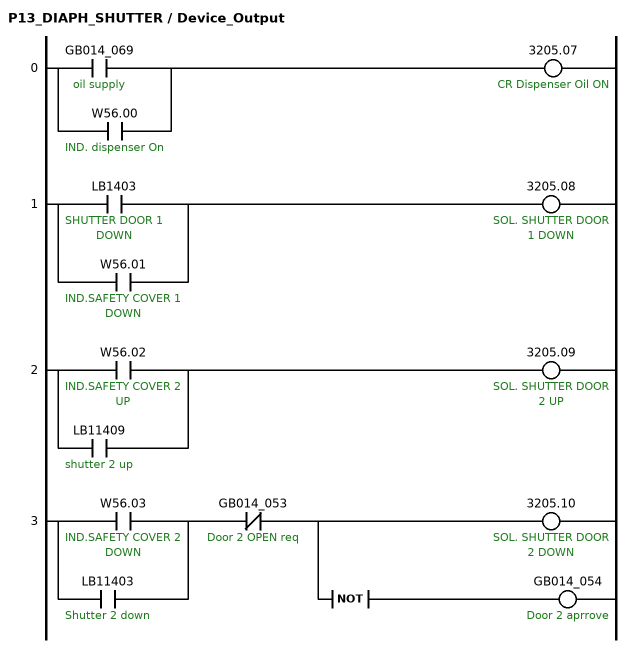
; [picture p168: P13_DIAPH_SHUTTER / Device_Output, rungs 0-3]
; rung 0
LD GB014_069  ; oil supply
OR W56.00  ; IND. dispenser On
OUT 3205.07  ; CR Dispenser Oil ON
; rung 1
LD LB1403  ; SHUTTER DOOR 1 DOWN
OR W56.01  ; IND.SAFETY COVER 1 DOWN
OUT 3205.08  ; SOL. SHUTTER DOOR 1 DOWN
; rung 2
LD W56.02  ; IND.SAFETY COVER 2 UP
OR LB11409  ; shutter 2 up
OUT 3205.09  ; SOL. SHUTTER DOOR 2 UP
; rung 3
LD W56.03  ; IND.SAFETY COVER 2 DOWN
OR LB11403  ; Shutter 2 down
ANDNOT GB014_053  ; Door 2 OPEN req
OUT 3205.10  ; SOL. SHUTTER DOOR 2 DOWN
NOT(520)
OUT GB014_054  ; Door 2 aprrove

### Section station_Output

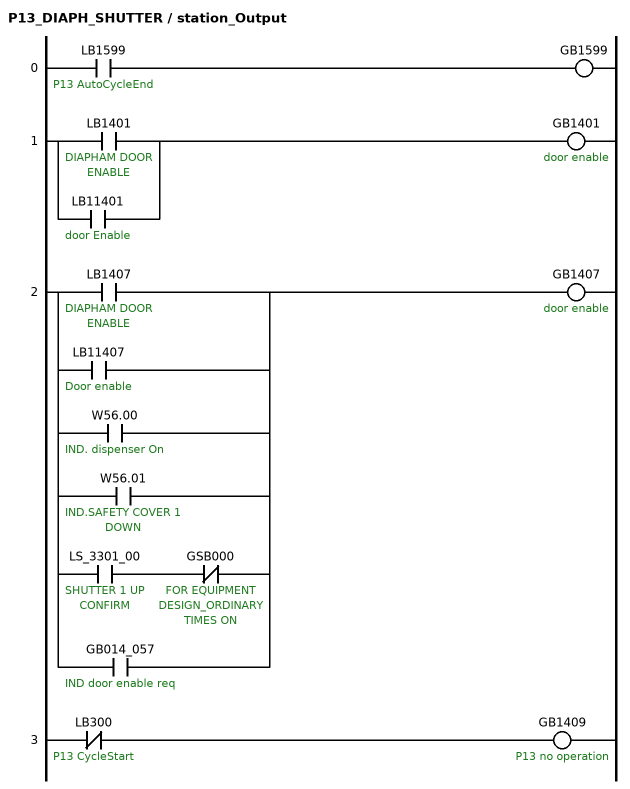
; rung 0
LD LB1599  ; P13 AutoCycleEnd
OUT GB1599
; rung 1
LD LB1401  ; DIAPHAM DOOR ENABLE
OR LB11401  ; door Enable
OUT GB1401  ; door enable
; rung 2
LD LB1407  ; DIAPHAM DOOR ENABLE
OR LB11407  ; Door enable
OR W56.00  ; IND. dispenser On
OR W56.01  ; IND.SAFETY COVER 1 DOWN
LD LS_3301_00  ; SHUTTER 1 UP CONFIRM
ANDNOT GSB000  ; FOR EQUIPMENT DESIGN_ORDINARY TIMES ON
ORLD
OR GB014_057  ; IND door enable req
OUT GB1407  ; door enable
; rung 3
LDNOT LB300  ; P13 CycleStart
OUT GB1409  ; P13 no operation

### Section END
; rung 0
END(001)

## Program P14_DIAPH_LOADER (cyclic task 4)
Local symbols
Disch_last_work E0_16.01 BOOL
Disch_last_work_operation_memory E0_16.02 BOOL
GB014_055 E0_45.06 BOOL  ; DOOR 2 OPEN req
GB014_056 E0_44.11 BOOL  ; IND door enable req
GB014_067 E0_42.12 BOOL  ; vacuum 1start
LB1000 E0_16.03 BOOL  ; AUTO START BEGIN
LB14234 E0_49.14 BOOL  ; oil supply motion
LB14235 E0_49.15 BOOL  ; oil supply finish
LB1600 E0_16.04 BOOL  ; AUTO START BEGIN
LB1601 E0_16.05 BOOL  ; 1EC3 FORWARD START
LB1601_1 E0_44.00 BOOL  ; EC4 backward
LB1601_12 E0_45.03 BOOL  ; Door 2 open req
LB1602 E0_16.06 BOOL  ; 1EC3 FORWARD START COMP
LB1602_1 E0_44.01 BOOL  ; EC4 bck conf
LB1603 E0_16.07 BOOL  ; GRIPPER UNIT DOWN
LB1604 E0_16.08 BOOL  ; GRIPPER UNIT DOWN CONF
LB1605 E0_16.09 BOOL  ; GRIPPER 1 DIAPH CHUCK
LB1606 E0_16.10 BOOL  ; GRIPPER 1 DIAPH CHUCK CONF
LB1607 E0_16.11 BOOL  ; GRIPPER UNIT UP
LB1608 E0_16.12 BOOL  ; GRIPPER UNIT UP CONF
LB1609 E0_16.13 BOOL  ; 1EC4 FORWARD START
LB1610 E0_16.14 BOOL  ; 1EC4 FORWARD START COMP
LB1611 E0_16.15 BOOL  ; 1EC3 MIDWARD START
LB16111 E0_17.00 BOOL  ; 1EC3 BACKWARD START
LB1612 E0_17.01 BOOL  ; 1EC3 FORWARD 2 START COMP
LB16121 E0_17.02 BOOL  ; 1EC3 BACKWARD START COMP
LB1612_1 E0_17.03 BOOL  ; flip 180
LB1612_2 E0_17.04 BOOL  ; Flip 180 confirm
LB1613 E0_17.05 BOOL  ; GRIPPER UNIT DOWN
LB1614 E0_17.06 BOOL  ; GRIPPER UNIT DOWN CONF
LB1615 E0_17.07 BOOL  ; GRIPPER 1 DIAPH UNCHUCK
LB1616 E0_17.08 BOOL  ; GRIPPER 1 DIAPH UNCHUCK CONF
LB1617 E0_17.09 BOOL  ; GRIPPER UNIT UP
LB1618 E0_17.10 BOOL  ; GRIPPER UNIT UP CONF
LB1618_1 E0_17.11 BOOL  ; Flip 0
LB1618_2 E0_17.12 BOOL  ; Flip 0 confirm
LB1619 E0_17.13 BOOL  ; 1EC4 BACKWARD START
LB1619_1 E0_44.13 BOOL  ; Door 2 open req
LB1620 E0_17.14 BOOL  ; 1EC4 BACKWARD START COMP
LB1621 E0_17.15 BOOL  ; 1EC3 BACKWARD START
LB1622 E0_18.00 BOOL  ; 1EC3 BACKWARD START COMP
LB1623 E0_18.01 BOOL  ; AUTO START BEGIN
LB1624 E0_18.02 BOOL  ; 1EC3 FORWARD START
LB1624_1 E0_44.02 BOOL  ; EC4 backward conf
LB1624_12 E0_45.04 BOOL  ; Door Open req
LB1625 E0_18.03 BOOL  ; 1EC3 FORWARD START COMP
LB1625_1 E0_44.03 BOOL  ; EC4 BCK confirm
LB1626 E0_18.04 BOOL  ; GRIPPER UNIT DOWN
LB1627 E0_18.05 BOOL  ; GRIPPER UNIT DOWN CONF
LB1628 E0_18.06 BOOL  ; GRIPPER 1 DIAPH CHUCK
LB1629 E0_18.07 BOOL  ; GRIPPER 1 DIAPH CHUCK CONF
LB1630 E0_18.08 BOOL  ; GRIPPER 2 DIAPH CHUCK
LB1631 E0_18.09 BOOL  ; GRIPPER 2 DIAPH CHUCK CONF
LB1632 E0_18.10 BOOL  ; GRIPPER UNIT UP
LB1633 E0_18.11 BOOL  ; GRIPPER UNIT UP CONF
LB1634 E0_18.12 BOOL  ; 1EC4 FORWARD START
LB1635 E0_18.13 BOOL  ; 1EC4 FORWARD START COMP
LB1636 E0_18.14 BOOL  ; 1EC3 MIDWARD START
LB16361 E0_18.15 BOOL  ; 1EC3 BACKWARD START
LB1637 E0_19.00 BOOL  ; 1EC3 FORWARD MID START COMP
LB16371 E0_19.01 BOOL  ; 1EC3 BACKWARD START COMP
LB16371_1 E0_19.02 BOOL  ; Rotate ADV
LB16371_2 E0_19.03 BOOL  ; Rotate ADV confirm
LB1639 E0_19.04 BOOL  ; GRIPPER UNIT DOWN
LB1640 E0_19.05 BOOL  ; GRIPPER UNIT DOWN CONF
LB1641 E0_19.06 BOOL  ; GRIPPER 1 DIAPH UNCHUCK
LB1642 E0_19.07 BOOL  ; GRIPPER 1 DIAPH UNCHUCK CONF
LB1643 E0_19.08 BOOL  ; GRIPPER 2 DIAPH UNCHUCK
LB1644 E0_19.09 BOOL  ; GRIPPER 2 DIAPH UNCHUCK CONF
LB1645 E0_19.10 BOOL  ; GRIPPER UNIT UP
LB1646 E0_19.11 BOOL  ; GRIPPER UNIT UP
LB1647 E0_19.12 BOOL  ; 1EC4 BACKWARD START
LB1647_1 E0_44.15 BOOL  ; door 2 req
LB1648 E0_19.13 BOOL  ; 1EC4 BACKWARD START COMP
LB1649 E0_19.14 BOOL  ; 1EC3 BACKWARD START
LB1650 E0_19.15 BOOL  ; 1EC3 BACKWARD START COMP
LB1650_1 E0_20.00 BOOL  ; Rotate return
LB1650_2 E0_20.01 BOOL  ; rotate ret confirm
LB1651 E0_20.02 BOOL  ; AUTO START BEGIN
LB1652 E0_20.03 BOOL  ; 1EC3 FORWARD START
LB1652_1 E0_44.05 BOOL  ; EC4 back
LB1652_12 E0_45.05 BOOL  ; Door open req
LB1653 E0_20.04 BOOL  ; 1EC3 FORWARD START COMP
LB1653_1 E0_44.04 BOOL  ; EC4 bck confirm
LB1654 E0_20.05 BOOL  ; GRIPPER UNIT DOWN
LB1655 E0_20.06 BOOL  ; GRIPPER UNIT DOWN CONF
LB1656 E0_20.07 BOOL  ; GRIPPER 1 DIAPH CHUCK
LB1657 E0_20.08 BOOL  ; GRIPPER 1 DIAPH CHUCK CONF
LB1658 E0_20.09 BOOL  ; GRIPPER 2 DIAPH CHUCK
LB1659 E0_20.10 BOOL  ; GRIPPER 2 DIAPH CHUCK CONF
LB1660 E0_20.11 BOOL  ; GRIPPER 3 DIAPH CHUCK
LB1661 E0_20.12 BOOL  ; GRIPPER 3 DIAPH CHUCK CONF
LB1662 E0_20.13 BOOL  ; GRIPPER UNIT UP
LB1663 E0_20.14 BOOL  ; GRIPPER UNIT UP CONF
LB1664 E0_20.15 BOOL  ; 1EC4 FORWARD START
LB1665 E0_21.00 BOOL  ; 1EC4 FORWARD START COMP
LB1666 E0_21.01 BOOL  ; 1EC3 MIDWARD START
LB16661 E0_21.02 BOOL  ; 1EC3 BACKWARD START
LB1667 E0_21.03 BOOL  ; 1EC3 FORWARD MID START COMP
LB16671 E0_21.04 BOOL  ; 1EC3 BACKWARD START COMP
LB1668 E0_21.05 BOOL  ; SOL.FILP DIAPH 180.
LB1669 E0_21.06 BOOL  ; SOL.FILP DIAPH 180. CONF
LB1670 E0_21.07 BOOL  ; GRIPPER UNIT DOWN
LB1670_1 E0_46.08 BOOL  ; cycle stop
LB1671 E0_21.08 BOOL  ; GRIPPER UNIT DOWN CONF
LB1672 E0_21.09 BOOL  ; GRIPPER 1 DIAPH UNCHUCK
LB1673 E0_21.10 BOOL  ; GRIPPER 1 DIAPH UNCHUCK CONF
LB1674 E0_21.11 BOOL  ; GRIPPER 2 DIAPH UNCHUCK
LB1675 E0_21.12 BOOL  ; GRIPPER 2 DIAPH UNCHUCK CONF
LB1676 E0_21.13 BOOL  ; GRIPPER 3 DIAPH UNCHUCK
LB1677 E0_21.14 BOOL  ; GRIPPER 3 DIAPH CONFUNCHUCK
LB1678 E0_21.15 BOOL  ; GRIPPER UNIT UP
LB1679 E0_22.00 BOOL  ; GRIPPER UNIT UP CONF
LB1680 E0_22.01 BOOL  ; 1EC4 BACKWARD START
LB1680_1 E0_45.02 BOOL  ; Door 2 open req
LB1681 E0_22.02 BOOL  ; 1EC4 BACKWARD START COMP
LB1682 E0_22.03 BOOL  ; 1EC3 BACKWARD START
LB1683 E0_22.04 BOOL  ; 1EC3 BACKWARD START COMP
LB1684 E0_22.05 BOOL  ; SOL.FILP DIAPH 0.
LB1685 E0_22.06 BOOL  ; SOL.FILP DIAPH 0. CONF
LB1686 E0_22.07 BOOL  ; AUTO START BEGIN
LB1687 E0_22.08 BOOL  ; GRIPPER UNIT DOWN
LB1688 E0_22.09 BOOL  ; GRIPPER UNIT DOWN CONF
LB1689 E0_22.10 BOOL  ; GRIPPER 3 DIAPH CHUCK
LB1690 E0_22.11 BOOL  ; GRIPPER 3 DIAPH CHUCK CONF
LB1691 E0_22.12 BOOL  ; GRIPPER UNIT UP
LB1692 E0_22.13 BOOL  ; GRIPPER UNIT UP CONF
LB1693 E0_22.14 BOOL  ; 1EC4 FORWARD START
LB1694 E0_22.15 BOOL  ; 1EC4 FORWARD START COMP
LB1695 E0_23.00 BOOL  ; 1EC3 MIDWARD START
LB16951 E0_23.01 BOOL  ; 1EC3 BACKWARD START
LB1696 E0_23.02 BOOL  ; 1EC3 FORWARD 2 START COMP
LB16961 E0_23.03 BOOL  ; 1EC3 BACKWARD START COMPL
LB1697 E0_23.04 BOOL  ; SOL.FILP DIAPH 180.
LB1698 E0_23.05 BOOL  ; SOL.FILP DIAPH 180. CONF
LB1699 E0_23.06 BOOL  ; GRIPPER UNIT DOWN
LB1700 E0_23.07 BOOL  ; GRIPPER UNIT DOWN CONF
LB1701 E0_23.08 BOOL  ; GRIPPER 3 DIAPH UNCHUCK
LB1702 E0_23.09 BOOL  ; GRIPPER 3 DIAPH UNCHUCK CONF
LB1703 E0_23.10 BOOL  ; GRIPPER UNIT UP
LB1704 E0_23.11 BOOL  ; GRIPPER UNIT UP CONF
LB1705 E0_23.12 BOOL  ; 1EC4 BACKWARD START
LB1705_1 E0_45.00 BOOL  ; door 2 open req
LB1706 E0_23.13 BOOL  ; 1EC4 BACKWARD START COMP
LB1707 E0_23.14 BOOL  ; 1EC3 BACKWARD START
LB1708 E0_23.15 BOOL  ; 1EC3 BACKWARD START COMP
LB1709 E0_24.00 BOOL  ; SOL.FILP DIAPH 0.
LB1710 E0_24.01 BOOL  ; SOL.FILP DIAPH 0. CONF
LB1711 E0_24.02 BOOL  ; AUTO START BEGIN
LB1712 E0_24.03 BOOL  ; GRIPPER UNIT DOWN
LB1713 E0_24.04 BOOL  ; GRIPPER UNIT DOWN CONF
LB1714 E0_24.05 BOOL  ; GRIPPER 2 DIAPH CHUCK
LB1715 E0_24.06 BOOL  ; GRIPPER 2 DIAPH CHUCK CONF
LB1716 E0_24.07 BOOL  ; GRIPPER 3 DIAPH CHUCK
LB1717 E0_24.08 BOOL  ; GRIPPER 3 DIAPH CHUCK CONF
LB1718 E0_24.09 BOOL  ; GRIPPER UNIT UP
LB1719 E0_24.10 BOOL  ; GRIPPER UNIT UP
LB1720 E0_24.11 BOOL  ; 1EC4 FORWARD START
LB1721 E0_24.12 BOOL  ; 1EC4 FORWARD START COMP
LB1724 E0_24.13 BOOL  ; SOL.FILP DIAPH 180.
LB1725 E0_24.14 BOOL  ; SOL.FILP DIAPH 180. CONF
LB1726 E0_24.15 BOOL  ; GRIPPER UNIT DOWN
LB1727 E0_25.00 BOOL  ; GRIPPER UNIT DOWN CONF
LB1728 E0_25.01 BOOL  ; GRIPPER 2 DIAPH UNCHUCK
LB1729 E0_25.02 BOOL  ; GRIPPER 2 DIAPH UNCHUCK CONF
LB1730 E0_25.03 BOOL  ; GRIPPER 3 DIAPH UNCHUCK
LB1731 E0_25.04 BOOL  ; GRIPPER 3 DIAPH CONFUNCHUCK
LB1732 E0_25.05 BOOL  ; GRIPPER UNIT UP
LB1733 E0_25.06 BOOL  ; GRIPPER UNIT UP CONF
LB1734 E0_25.07 BOOL  ; 1EC4 BACKWARD START
LB1734_1 E0_45.01 BOOL  ; Door 2 open req
LB1735 E0_25.08 BOOL  ; 1EC4 BACKWARD START COMP
LB1736 E0_25.09 BOOL  ; SOL.FILP DIAPH 0.
LB1737 E0_25.10 BOOL  ; SOL.FILP DIAPH 0. CONF
LB1791 E0_25.11 BOOL  ; P14  Case1 End
LB1792 E0_25.12 BOOL  ; P14  Case2 End
LB1793 E0_25.13 BOOL  ; P14  Case3 End
LB1794 E0_25.14 BOOL  ; P14  Case4 End
LB1795 E0_25.15 BOOL  ; P14  Case5 End
LB1799 E0_26.00 BOOL  ; P14 AutoCycleEnd
LB324 E0_49.13 BOOL  ; oil supply condition
LB340 E0_26.01 BOOL  ; IND 1 CYCLE
LB400 E0_26.02 BOOL  ; P14 CycleStart
LB401 E0_26.03 BOOL  ; P14 LoadIn Case1
LB402 E0_26.04 BOOL  ; P14 LoadIn Case2
LB403 E0_26.05 BOOL  ; P14 LoadIn Case3
LB404 E0_26.06 BOOL  ; P14 LoadIn Case4(DisCH)
LB405 E0_26.07 BOOL  ; P14 LoadIn Case5(DisCH)
LB406 E0_26.08 BOOL  ; P14 UnLoad Case1
LB407 E0_26.09 BOOL  ; P14 UnLoad Case2
LB408 E0_26.10 BOOL  ; P14 UnLoad Case3
LB409 E0_26.11 BOOL  ; P14 UnLoad Case4(DisCH)
LB410 E0_26.12 BOOL  ; P14 UnLoad Case5(DisCH)
LB560 E0_44.07 BOOL  ; DOOR ENABLE req
LB5600 E0_44.10 BOOL  ; Door enable req
LB5601 E0_44.06 BOOL  ; DOOR ENABLE REq
LB5602 E0_44.08 BOOL  ; DOOR ENABLE REQ
LB5603 E0_44.09 BOOL  ; DOOR enable req
LD213 E0_50 UINT  ; memory count
LT3234 T3043 TIMER
LT4355 E0_51.00 BOOL
LT4356 T3044 TIMER
LT876 T3035 TIMER
Stopwatch1 E0_27 DINT
Stopwatch2 E0_29 UINT
dbug E0_26.13 BOOL
p_oN E0_49.11 BOOL

### Section HMI_Output

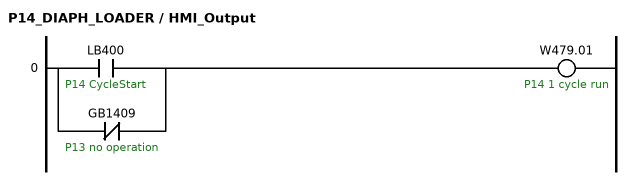
; rung 0
LD LB400  ; P14 CycleStart
ORNOT GB1409  ; P13 no operation
OUT W479.01  ; P14 1 cycle run

### Section Condition

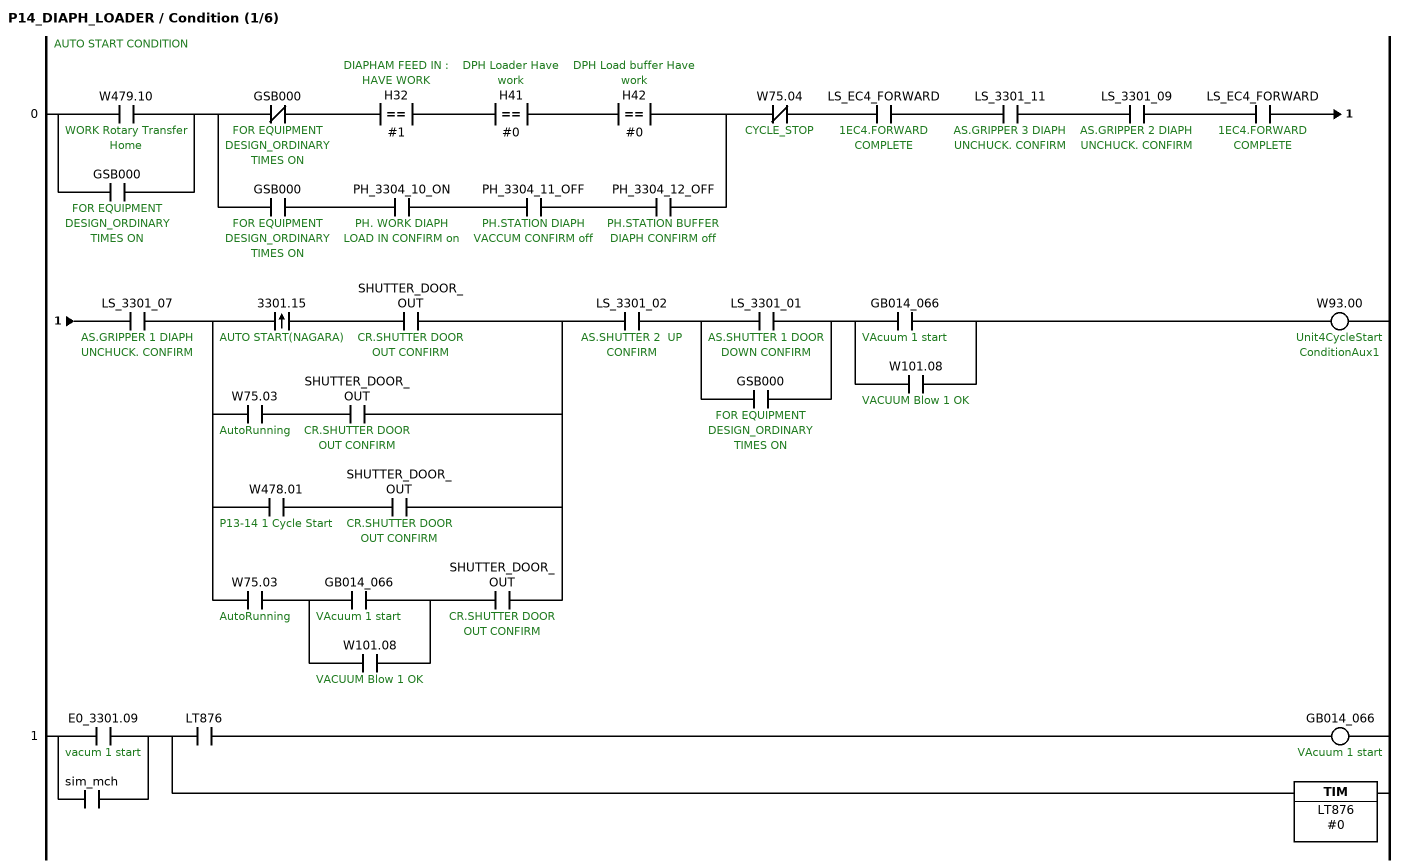
; rung 0: AUTO START CONDITION
LD W479.10  ; WORK Rotary Transfer Home
OR GSB000  ; FOR EQUIPMENT DESIGN_ORDINARY TIMES ON
LDNOT GSB000  ; FOR EQUIPMENT DESIGN_ORDINARY TIMES ON
AND=(300) H32 #1  ; DIAPHAM FEED IN : HAVE WORK
AND=(300) H41 #0  ; DPH Loader Have work
AND=(300) H42 #0  ; DPH Load buffer Have work
LD GSB000  ; FOR EQUIPMENT DESIGN_ORDINARY TIMES ON
AND PH_3304_10_ON  ; PH. WORK DIAPH LOAD IN CONFIRM on
AND PH_3304_11_OFF  ; PH.STATION DIAPH VACCUM CONFIRM off
AND PH_3304_12_OFF  ; PH.STATION BUFFER DIAPH CONFIRM off
ORLD
ANDLD
ANDNOT W75.04  ; CYCLE_STOP
AND LS_EC4_FORWARD  ; 1EC4.FORWARD COMPLETE
AND LS_3301_11  ; AS.GRIPPER 3 DIAPH UNCHUCK. CONFIRM
AND LS_3301_09  ; AS.GRIPPER 2 DIAPH UNCHUCK. CONFIRM
AND LS_EC4_FORWARD  ; 1EC4.FORWARD COMPLETE
AND LS_3301_07  ; AS.GRIPPER 1 DIAPH UNCHUCK. CONFIRM
@LD 3301.15  ; AUTO START(NAGARA)
AND SHUTTER_DOOR_OUT  ; CR.SHUTTER DOOR OUT CONFIRM
LD W75.03  ; AutoRunning
AND SHUTTER_DOOR_OUT  ; CR.SHUTTER DOOR OUT CONFIRM
ORLD
LD W478.01  ; P13-14 1 Cycle Start
AND SHUTTER_DOOR_OUT  ; CR.SHUTTER DOOR OUT CONFIRM
ORLD
LD W75.03  ; AutoRunning
LD GB014_066  ; VAcuum 1 start
OR W101.08  ; VACUUM Blow 1 OK
ANDLD
AND SHUTTER_DOOR_OUT  ; CR.SHUTTER DOOR OUT CONFIRM
ORLD
ANDLD
AND LS_3301_02  ; AS.SHUTTER 2  UP CONFIRM
LD LS_3301_01  ; AS.SHUTTER 1 DOOR DOWN CONFIRM
OR GSB000  ; FOR EQUIPMENT DESIGN_ORDINARY TIMES ON
ANDLD
LD GB014_066  ; VAcuum 1 start
OR W101.08  ; VACUUM Blow 1 OK
ANDLD
OUT W93.00  ; Unit4CycleStartConditionAux1
; rung 1
LD E0_3301.09  ; vacum 1 start
OR sim_mch
OUT TR0
AND LT876
OUT GB014_066  ; VAcuum 1 start
LD TR0
TIM LT876 #0

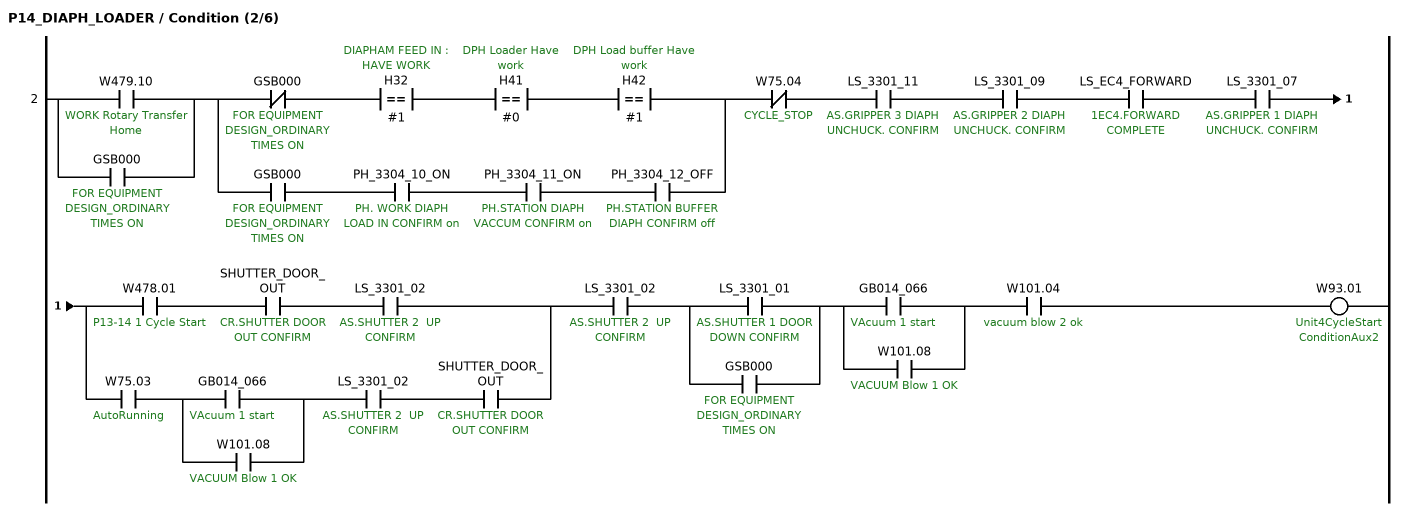
; rung 2
LD W479.10  ; WORK Rotary Transfer Home
OR GSB000  ; FOR EQUIPMENT DESIGN_ORDINARY TIMES ON
LDNOT GSB000  ; FOR EQUIPMENT DESIGN_ORDINARY TIMES ON
AND=(300) H32 #1  ; DIAPHAM FEED IN : HAVE WORK
AND=(300) H41 #0  ; DPH Loader Have work
AND=(300) H42 #1  ; DPH Load buffer Have work
LD GSB000  ; FOR EQUIPMENT DESIGN_ORDINARY TIMES ON
AND PH_3304_10_ON  ; PH. WORK DIAPH LOAD IN CONFIRM on
AND PH_3304_11_ON  ; PH.STATION DIAPH VACCUM CONFIRM on
AND PH_3304_12_OFF  ; PH.STATION BUFFER DIAPH CONFIRM off
ORLD
ANDLD
ANDNOT W75.04  ; CYCLE_STOP
AND LS_3301_11  ; AS.GRIPPER 3 DIAPH UNCHUCK. CONFIRM
AND LS_3301_09  ; AS.GRIPPER 2 DIAPH UNCHUCK. CONFIRM
AND LS_EC4_FORWARD  ; 1EC4.FORWARD COMPLETE
AND LS_3301_07  ; AS.GRIPPER 1 DIAPH UNCHUCK. CONFIRM
LD W478.01  ; P13-14 1 Cycle Start
AND SHUTTER_DOOR_OUT  ; CR.SHUTTER DOOR OUT CONFIRM
AND LS_3301_02  ; AS.SHUTTER 2  UP CONFIRM
LD W75.03  ; AutoRunning
LD GB014_066  ; VAcuum 1 start
OR W101.08  ; VACUUM Blow 1 OK
ANDLD
AND LS_3301_02  ; AS.SHUTTER 2  UP CONFIRM
AND SHUTTER_DOOR_OUT  ; CR.SHUTTER DOOR OUT CONFIRM
ORLD
ANDLD
AND LS_3301_02  ; AS.SHUTTER 2  UP CONFIRM
LD LS_3301_01  ; AS.SHUTTER 1 DOOR DOWN CONFIRM
OR GSB000  ; FOR EQUIPMENT DESIGN_ORDINARY TIMES ON
ANDLD
LD GB014_066  ; VAcuum 1 start
OR W101.08  ; VACUUM Blow 1 OK
ANDLD
AND W101.04  ; vacuum blow 2 ok
OUT W93.01  ; Unit4CycleStartConditionAux2

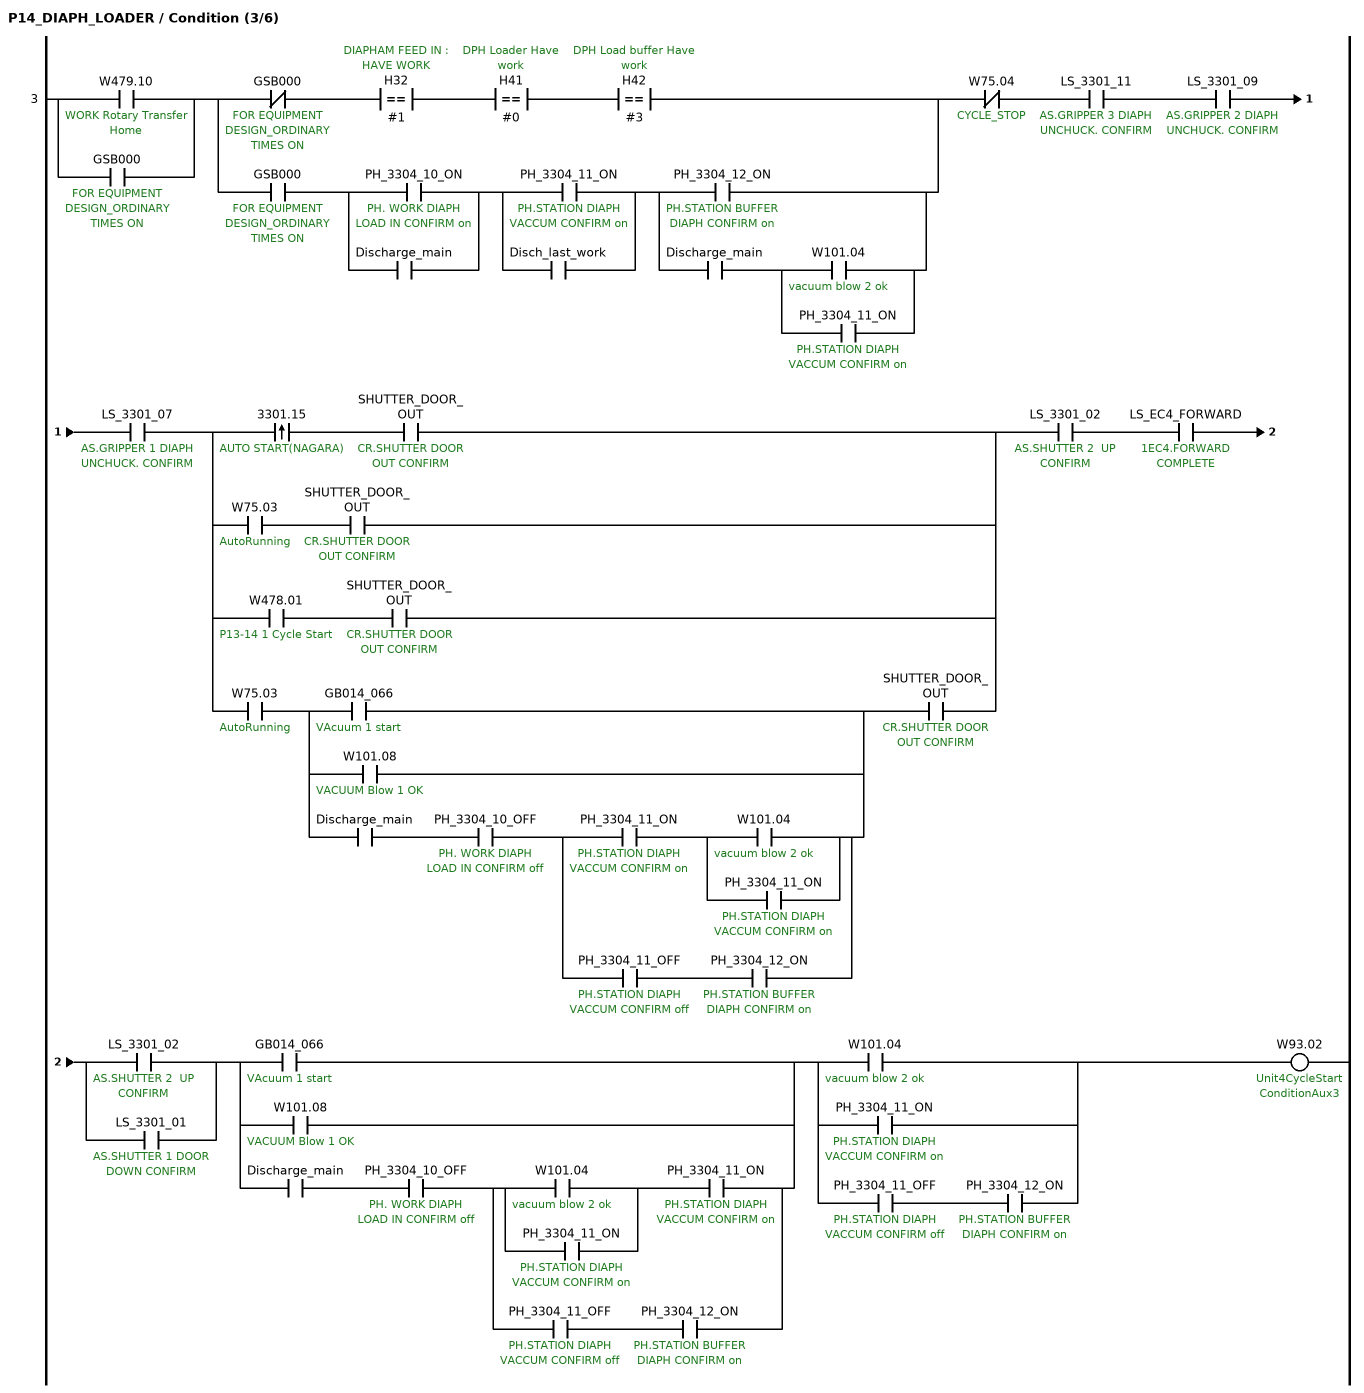
; rung 3
LD W479.10  ; WORK Rotary Transfer Home
OR GSB000  ; FOR EQUIPMENT DESIGN_ORDINARY TIMES ON
LDNOT GSB000  ; FOR EQUIPMENT DESIGN_ORDINARY TIMES ON
AND=(300) H32 #1  ; DIAPHAM FEED IN : HAVE WORK
AND=(300) H41 #0  ; DPH Loader Have work
AND=(300) H42 #3  ; DPH Load buffer Have work
LD GSB000  ; FOR EQUIPMENT DESIGN_ORDINARY TIMES ON
LD PH_3304_10_ON  ; PH. WORK DIAPH LOAD IN CONFIRM on
OR Discharge_main
ANDLD
LD PH_3304_11_ON  ; PH.STATION DIAPH VACCUM CONFIRM on
OR Disch_last_work
ANDLD
LD PH_3304_12_ON  ; PH.STATION BUFFER DIAPH CONFIRM on
LD Discharge_main
LD W101.04  ; vacuum blow 2 ok
OR PH_3304_11_ON  ; PH.STATION DIAPH VACCUM CONFIRM on
ANDLD
ORLD
ANDLD
ORLD
ANDLD
ANDNOT W75.04  ; CYCLE_STOP
AND LS_3301_11  ; AS.GRIPPER 3 DIAPH UNCHUCK. CONFIRM
AND LS_3301_09  ; AS.GRIPPER 2 DIAPH UNCHUCK. CONFIRM
AND LS_3301_07  ; AS.GRIPPER 1 DIAPH UNCHUCK. CONFIRM
@LD 3301.15  ; AUTO START(NAGARA)
AND SHUTTER_DOOR_OUT  ; CR.SHUTTER DOOR OUT CONFIRM
LD W75.03  ; AutoRunning
AND SHUTTER_DOOR_OUT  ; CR.SHUTTER DOOR OUT CONFIRM
ORLD
LD W478.01  ; P13-14 1 Cycle Start
AND SHUTTER_DOOR_OUT  ; CR.SHUTTER DOOR OUT CONFIRM
ORLD
LD W75.03  ; AutoRunning
LD GB014_066  ; VAcuum 1 start
OR W101.08  ; VACUUM Blow 1 OK
LD Discharge_main
AND PH_3304_10_OFF  ; PH. WORK DIAPH LOAD IN CONFIRM off
LD PH_3304_11_ON  ; PH.STATION DIAPH VACCUM CONFIRM on
LD W101.04  ; vacuum blow 2 ok
OR PH_3304_11_ON  ; PH.STATION DIAPH VACCUM CONFIRM on
ANDLD
LD PH_3304_11_OFF  ; PH.STATION DIAPH VACCUM CONFIRM off
AND PH_3304_12_ON  ; PH.STATION BUFFER DIAPH CONFIRM on
ORLD
ANDLD
ORLD
ANDLD
AND SHUTTER_DOOR_OUT  ; CR.SHUTTER DOOR OUT CONFIRM
ORLD
ANDLD
AND LS_3301_02  ; AS.SHUTTER 2  UP CONFIRM
AND LS_EC4_FORWARD  ; 1EC4.FORWARD COMPLETE
LD LS_3301_02  ; AS.SHUTTER 2  UP CONFIRM
OR LS_3301_01  ; AS.SHUTTER 1 DOOR DOWN CONFIRM
ANDLD
LD GB014_066  ; VAcuum 1 start
OR W101.08  ; VACUUM Blow 1 OK
LD Discharge_main
AND PH_3304_10_OFF  ; PH. WORK DIAPH LOAD IN CONFIRM off
LD W101.04  ; vacuum blow 2 ok
OR PH_3304_11_ON  ; PH.STATION DIAPH VACCUM CONFIRM on
AND PH_3304_11_ON  ; PH.STATION DIAPH VACCUM CONFIRM on
LD PH_3304_11_OFF  ; PH.STATION DIAPH VACCUM CONFIRM off
AND PH_3304_12_ON  ; PH.STATION BUFFER DIAPH CONFIRM on
ORLD
ANDLD
ORLD
ANDLD
LD W101.04  ; vacuum blow 2 ok
OR PH_3304_11_ON  ; PH.STATION DIAPH VACCUM CONFIRM on
LD PH_3304_11_OFF  ; PH.STATION DIAPH VACCUM CONFIRM off
AND PH_3304_12_ON  ; PH.STATION BUFFER DIAPH CONFIRM on
ORLD
ANDLD
OUT W93.02  ; Unit4CycleStartConditionAux3

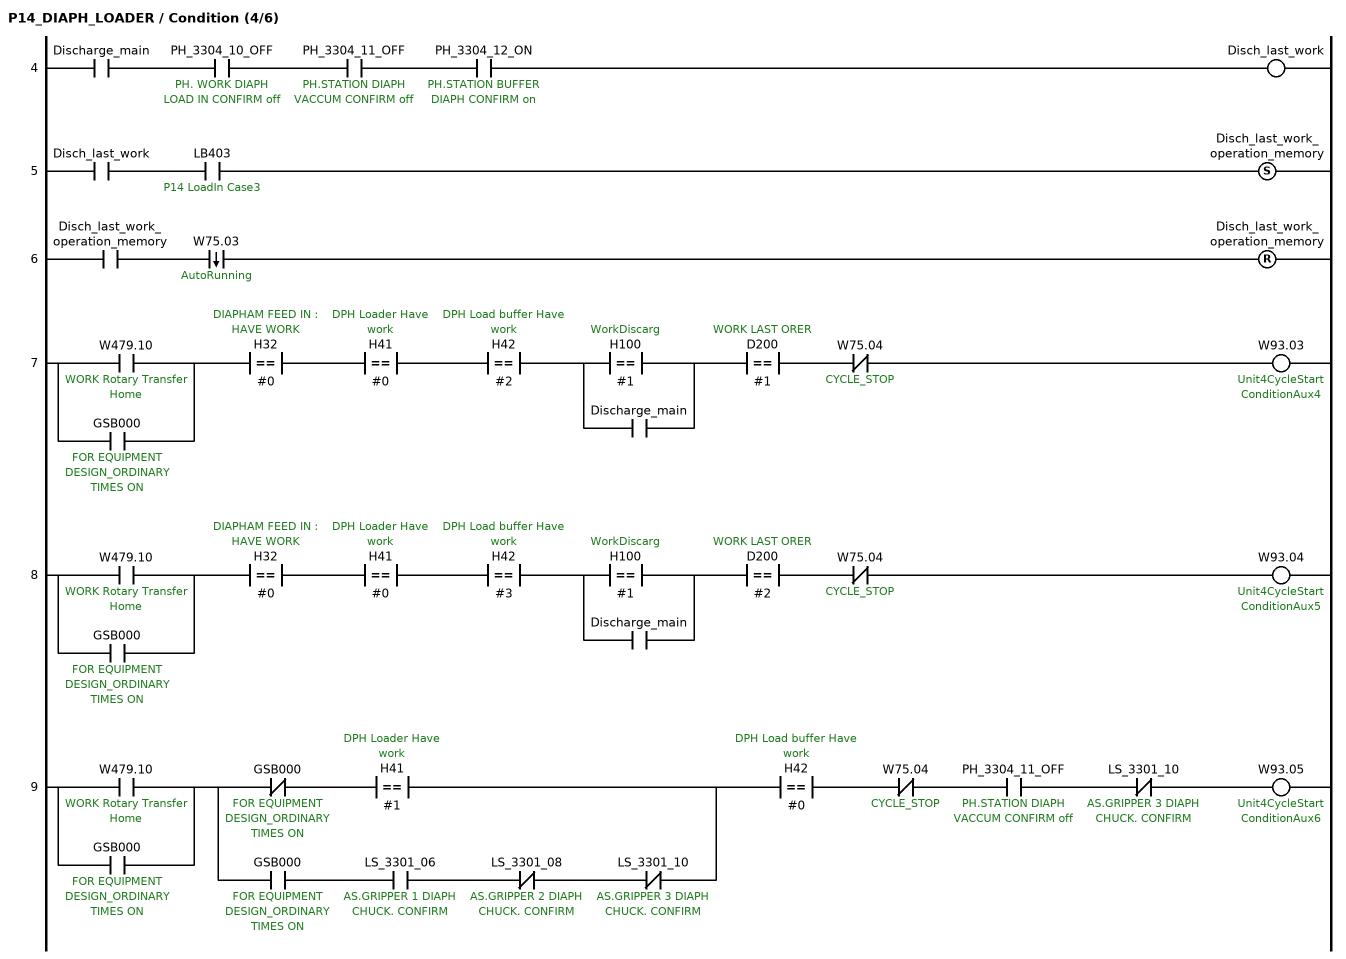
; rung 4
LD Discharge_main
AND PH_3304_10_OFF  ; PH. WORK DIAPH LOAD IN CONFIRM off
AND PH_3304_11_OFF  ; PH.STATION DIAPH VACCUM CONFIRM off
AND PH_3304_12_ON  ; PH.STATION BUFFER DIAPH CONFIRM on
OUT Disch_last_work
; rung 5
LD Disch_last_work
AND LB403  ; P14 LoadIn Case3
SET Disch_last_work_operation_memory
; rung 6
LD Disch_last_work_operation_memory
%AND W75.03  ; AutoRunning
RSET Disch_last_work_operation_memory
; rung 7
LD W479.10  ; WORK Rotary Transfer Home
OR GSB000  ; FOR EQUIPMENT DESIGN_ORDINARY TIMES ON
AND=(300) H32 #0  ; DIAPHAM FEED IN : HAVE WORK
AND=(300) H41 #0  ; DPH Loader Have work
AND=(300) H42 #2  ; DPH Load buffer Have work
LD=(300) H100 #1  ; WorkDiscarg
OR Discharge_main
ANDLD
AND=(300) D200 #1  ; WORK LAST ORER
ANDNOT W75.04  ; CYCLE_STOP
OUT W93.03  ; Unit4CycleStartConditionAux4
; rung 8
LD W479.10  ; WORK Rotary Transfer Home
OR GSB000  ; FOR EQUIPMENT DESIGN_ORDINARY TIMES ON
AND=(300) H32 #0  ; DIAPHAM FEED IN : HAVE WORK
AND=(300) H41 #0  ; DPH Loader Have work
AND=(300) H42 #3  ; DPH Load buffer Have work
LD=(300) H100 #1  ; WorkDiscarg
OR Discharge_main
ANDLD
AND=(300) D200 #2  ; WORK LAST ORER
ANDNOT W75.04  ; CYCLE_STOP
OUT W93.04  ; Unit4CycleStartConditionAux5
; rung 9
LD W479.10  ; WORK Rotary Transfer Home
OR GSB000  ; FOR EQUIPMENT DESIGN_ORDINARY TIMES ON
LDNOT GSB000  ; FOR EQUIPMENT DESIGN_ORDINARY TIMES ON
AND=(300) H41 #1  ; DPH Loader Have work
LD GSB000  ; FOR EQUIPMENT DESIGN_ORDINARY TIMES ON
AND LS_3301_06  ; AS.GRIPPER 1 DIAPH CHUCK. CONFIRM
ANDNOT LS_3301_08  ; AS.GRIPPER 2 DIAPH CHUCK. CONFIRM
ANDNOT LS_3301_10  ; AS.GRIPPER 3 DIAPH CHUCK. CONFIRM
ORLD
ANDLD
AND=(300) H42 #0  ; DPH Load buffer Have work
ANDNOT W75.04  ; CYCLE_STOP
AND PH_3304_11_OFF  ; PH.STATION DIAPH VACCUM CONFIRM off
ANDNOT LS_3301_10  ; AS.GRIPPER 3 DIAPH CHUCK. CONFIRM
OUT W93.05  ; Unit4CycleStartConditionAux6

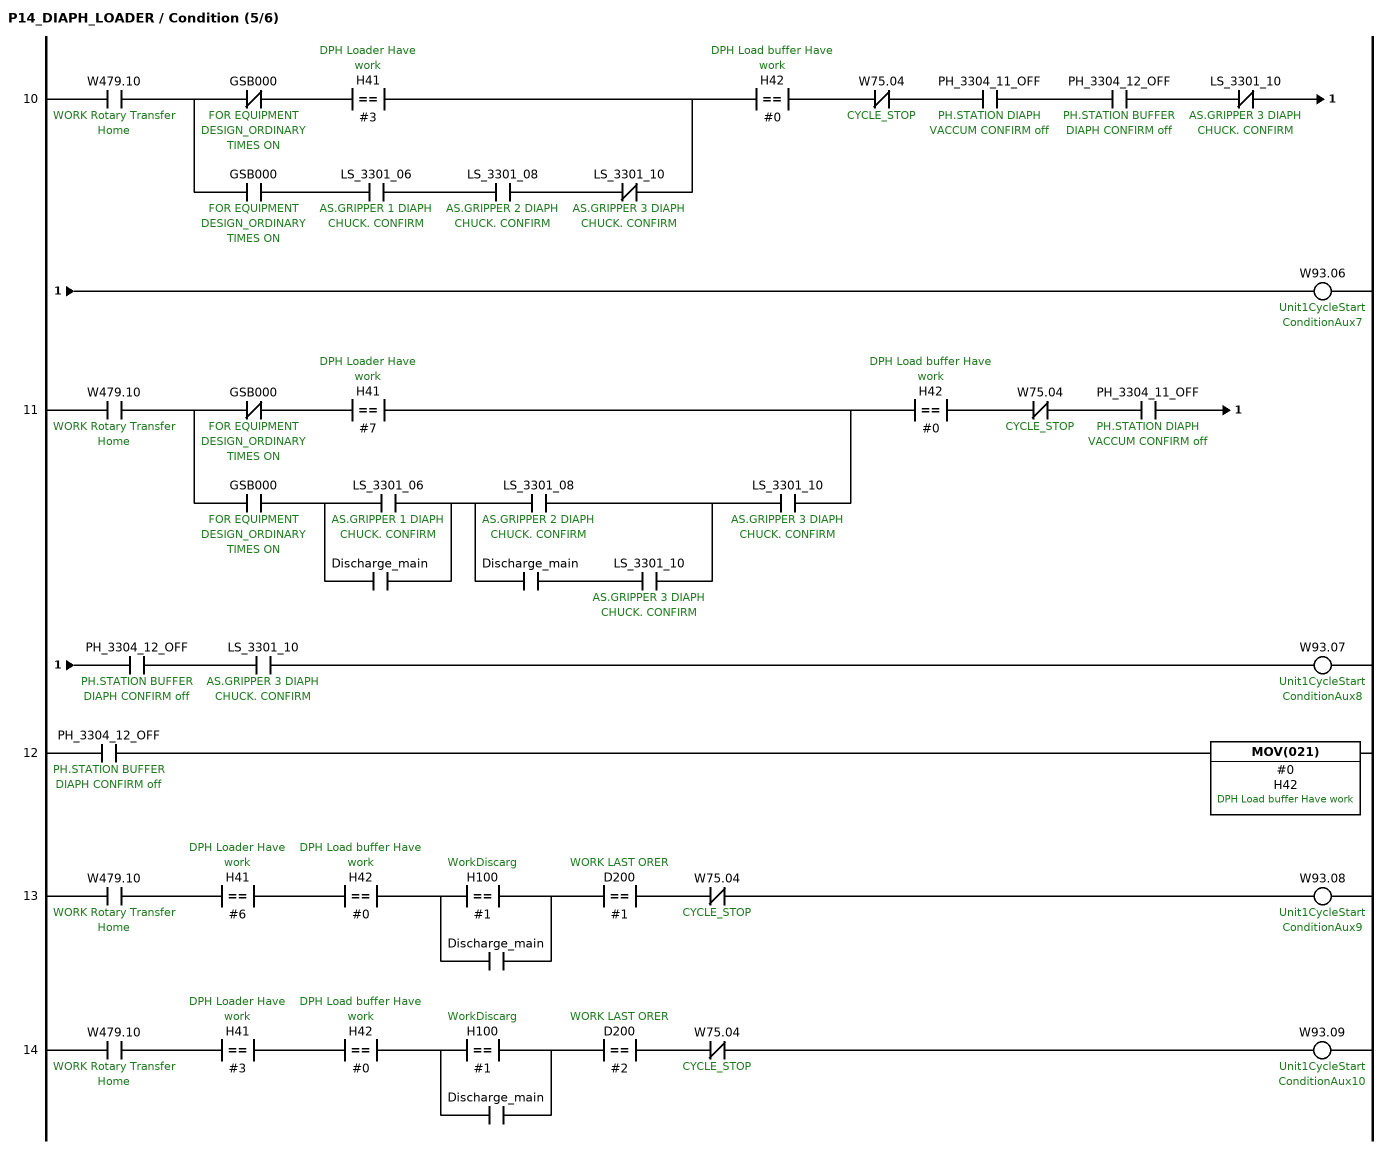
; rung 10
LD W479.10  ; WORK Rotary Transfer Home
LDNOT GSB000  ; FOR EQUIPMENT DESIGN_ORDINARY TIMES ON
AND=(300) H41 #3  ; DPH Loader Have work
LD GSB000  ; FOR EQUIPMENT DESIGN_ORDINARY TIMES ON
AND LS_3301_06  ; AS.GRIPPER 1 DIAPH CHUCK. CONFIRM
AND LS_3301_08  ; AS.GRIPPER 2 DIAPH CHUCK. CONFIRM
ANDNOT LS_3301_10  ; AS.GRIPPER 3 DIAPH CHUCK. CONFIRM
ORLD
ANDLD
AND=(300) H42 #0  ; DPH Load buffer Have work
ANDNOT W75.04  ; CYCLE_STOP
AND PH_3304_11_OFF  ; PH.STATION DIAPH VACCUM CONFIRM off
AND PH_3304_12_OFF  ; PH.STATION BUFFER DIAPH CONFIRM off
ANDNOT LS_3301_10  ; AS.GRIPPER 3 DIAPH CHUCK. CONFIRM
OUT W93.06  ; Unit1CycleStartConditionAux7
; rung 11
LD W479.10  ; WORK Rotary Transfer Home
LDNOT GSB000  ; FOR EQUIPMENT DESIGN_ORDINARY TIMES ON
AND=(300) H41 #7  ; DPH Loader Have work
LD GSB000  ; FOR EQUIPMENT DESIGN_ORDINARY TIMES ON
LD LS_3301_06  ; AS.GRIPPER 1 DIAPH CHUCK. CONFIRM
OR Discharge_main
ANDLD
LD LS_3301_08  ; AS.GRIPPER 2 DIAPH CHUCK. CONFIRM
LD Discharge_main
AND LS_3301_10  ; AS.GRIPPER 3 DIAPH CHUCK. CONFIRM
ORLD
ANDLD
AND LS_3301_10  ; AS.GRIPPER 3 DIAPH CHUCK. CONFIRM
ORLD
ANDLD
AND=(300) H42 #0  ; DPH Load buffer Have work
ANDNOT W75.04  ; CYCLE_STOP
AND PH_3304_11_OFF  ; PH.STATION DIAPH VACCUM CONFIRM off
AND PH_3304_12_OFF  ; PH.STATION BUFFER DIAPH CONFIRM off
AND LS_3301_10  ; AS.GRIPPER 3 DIAPH CHUCK. CONFIRM
OUT W93.07  ; Unit1CycleStartConditionAux8
; rung 12
LD PH_3304_12_OFF  ; PH.STATION BUFFER DIAPH CONFIRM off
MOV(021) #0 H42  ; DPH Load buffer Have work
; rung 13
LD W479.10  ; WORK Rotary Transfer Home
AND=(300) H41 #6  ; DPH Loader Have work
AND=(300) H42 #0  ; DPH Load buffer Have work
LD=(300) H100 #1  ; WorkDiscarg
OR Discharge_main
ANDLD
AND=(300) D200 #1  ; WORK LAST ORER
ANDNOT W75.04  ; CYCLE_STOP
OUT W93.08  ; Unit1CycleStartConditionAux9
; rung 14
LD W479.10  ; WORK Rotary Transfer Home
AND=(300) H41 #3  ; DPH Loader Have work
AND=(300) H42 #0  ; DPH Load buffer Have work
LD=(300) H100 #1  ; WorkDiscarg
OR Discharge_main
ANDLD
AND=(300) D200 #2  ; WORK LAST ORER
ANDNOT W75.04  ; CYCLE_STOP
OUT W93.09  ; Unit1CycleStartConditionAux10

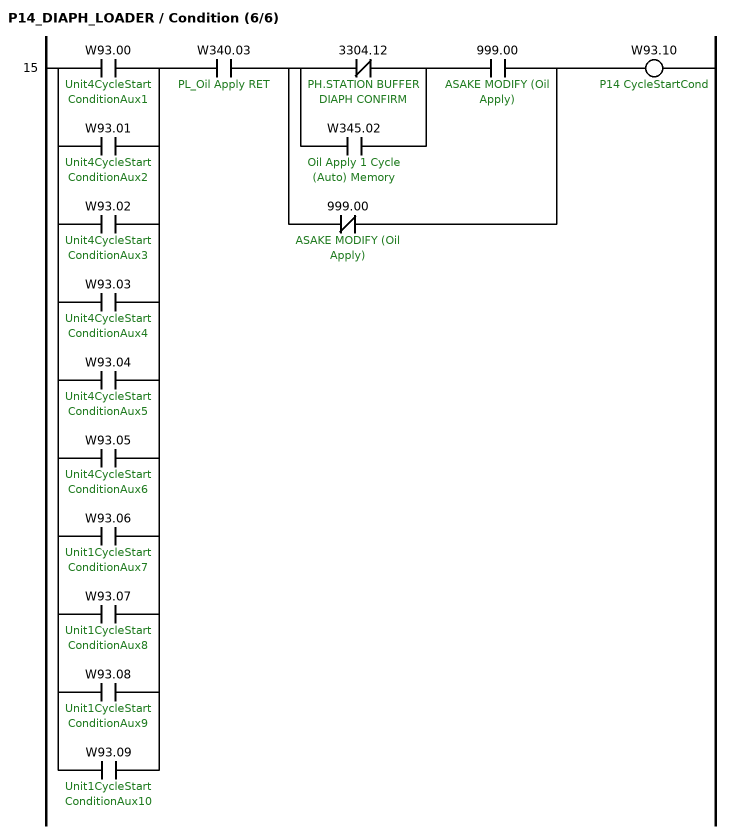
; rung 15
LD W93.00  ; Unit4CycleStartConditionAux1
OR W93.01  ; Unit4CycleStartConditionAux2
OR W93.02  ; Unit4CycleStartConditionAux3
OR W93.03  ; Unit4CycleStartConditionAux4
OR W93.04  ; Unit4CycleStartConditionAux5
OR W93.05  ; Unit4CycleStartConditionAux6
OR W93.06  ; Unit1CycleStartConditionAux7
OR W93.07  ; Unit1CycleStartConditionAux8
OR W93.08  ; Unit1CycleStartConditionAux9
OR W93.09  ; Unit1CycleStartConditionAux10
AND W340.03  ; PL_Oil Apply RET
LDNOT 3304.12  ; PH.STATION BUFFER DIAPH CONFIRM
OR W345.02  ; Oil Apply 1 Cycle (Auto) Memory
AND 999.00  ; ASAKE MODIFY (Oil Apply)
ORNOT 999.00  ; ASAKE MODIFY (Oil Apply)
ANDLD
OUT W93.10  ; P14 CycleStartCond

### Section Autorun

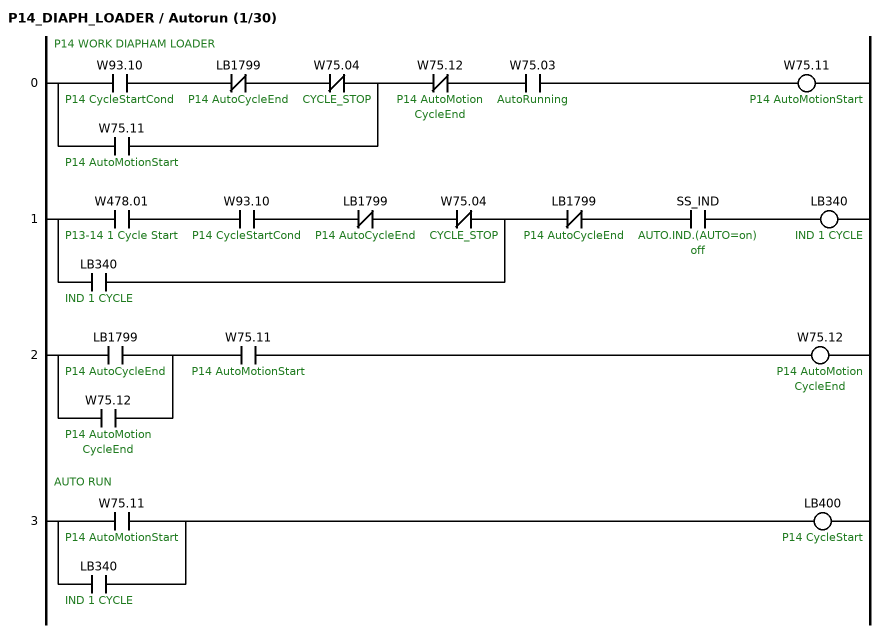
; rung 0: P14 WORK DIAPHAM LOADER
LD W93.10  ; P14 CycleStartCond
ANDNOT LB1799  ; P14 AutoCycleEnd
ANDNOT W75.04  ; CYCLE_STOP
OR W75.11  ; P14 AutoMotionStart
ANDNOT W75.12  ; P14 AutoMotion CycleEnd
AND W75.03  ; AutoRunning
OUT W75.11  ; P14 AutoMotionStart
; rung 1
LD W478.01  ; P13-14 1 Cycle Start
AND W93.10  ; P14 CycleStartCond
ANDNOT LB1799  ; P14 AutoCycleEnd
ANDNOT W75.04  ; CYCLE_STOP
OR LB340  ; IND 1 CYCLE
ANDNOT LB1799  ; P14 AutoCycleEnd
AND SS_IND  ; AUTO.IND.(AUTO=on) off
OUT LB340  ; IND 1 CYCLE
; rung 2
LD LB1799  ; P14 AutoCycleEnd
OR W75.12  ; P14 AutoMotion CycleEnd
AND W75.11  ; P14 AutoMotionStart
OUT W75.12  ; P14 AutoMotion CycleEnd
; rung 3: AUTO RUN
LD W75.11  ; P14 AutoMotionStart
OR LB340  ; IND 1 CYCLE
OUT LB400  ; P14 CycleStart

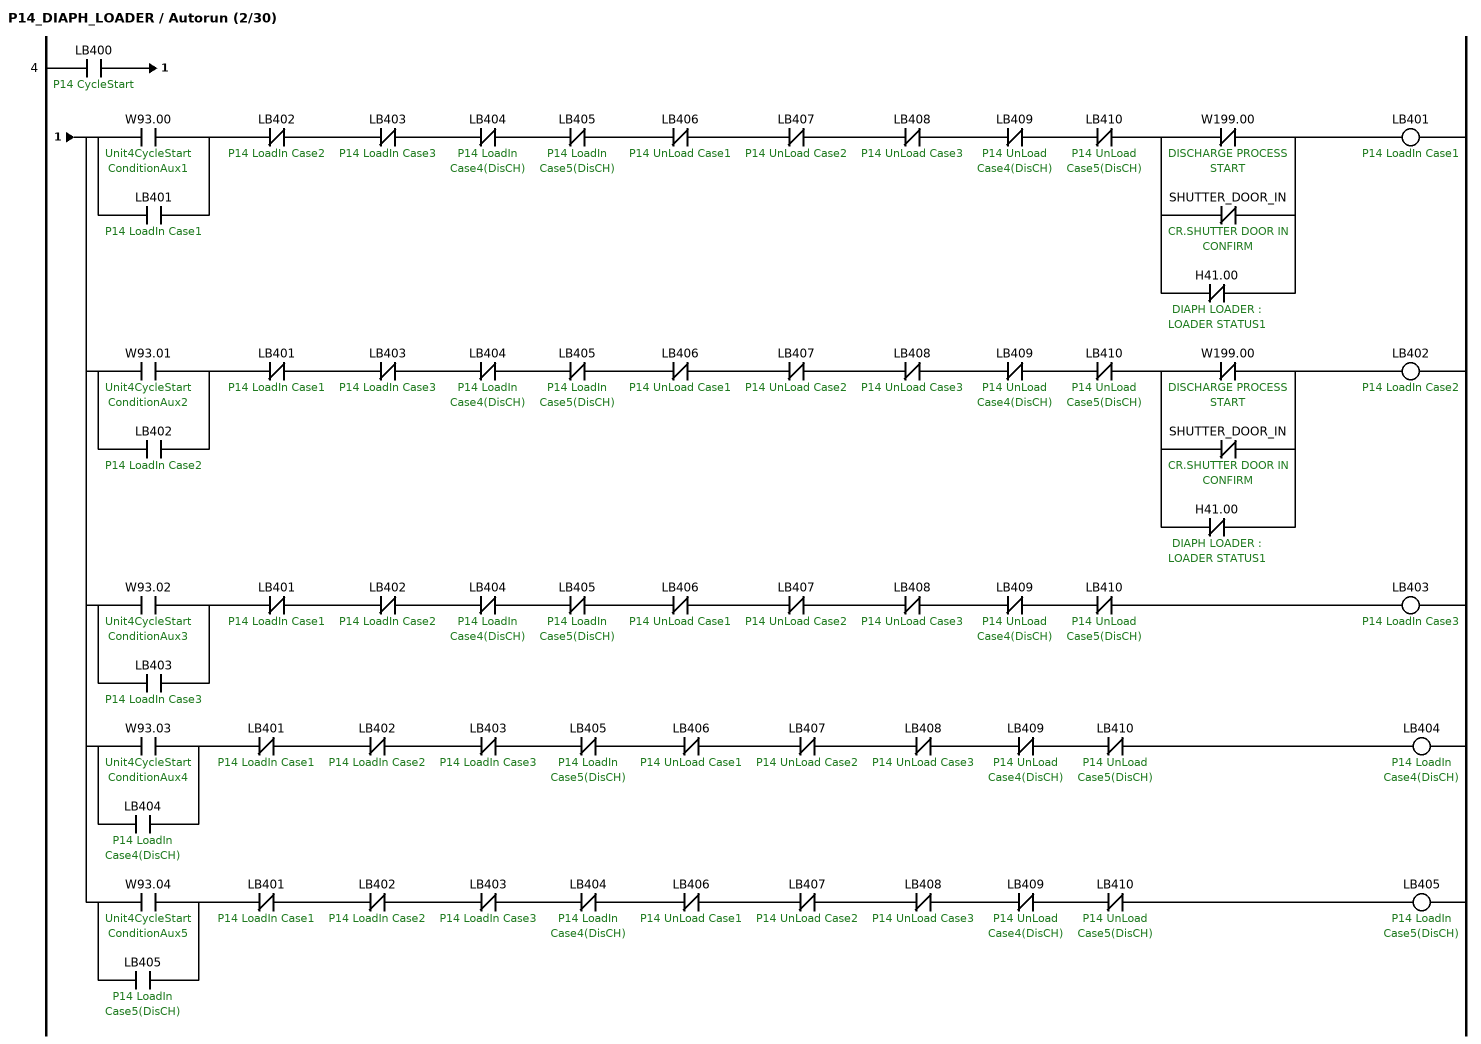
; rung 4
LD LB400  ; P14 CycleStart
OUT TR0
LD W93.00  ; Unit4CycleStartConditionAux1
OR LB401  ; P14 LoadIn Case1
ANDLD
ANDNOT LB402  ; P14 LoadIn Case2
ANDNOT LB403  ; P14 LoadIn Case3
ANDNOT LB404  ; P14 LoadIn Case4(DisCH)
ANDNOT LB405  ; P14 LoadIn Case5(DisCH)
ANDNOT LB406  ; P14 UnLoad Case1
ANDNOT LB407  ; P14 UnLoad Case2
ANDNOT LB408  ; P14 UnLoad Case3
ANDNOT LB409  ; P14 UnLoad Case4(DisCH)
ANDNOT LB410  ; P14 UnLoad Case5(DisCH)
LDNOT W199.00  ; DISCHARGE PROCESS START  // To protect conflict loop from dummy
ORNOT SHUTTER_DOOR_IN  ; CR.SHUTTER DOOR IN CONFIRM
ORNOT H41.00  ; DIAPH LOADER : LOADER STATUS1
ANDLD
OUT LB401  ; P14 LoadIn Case1
LD TR0
LD W93.01  ; Unit4CycleStartConditionAux2
OR LB402  ; P14 LoadIn Case2
ANDLD
ANDNOT LB401  ; P14 LoadIn Case1
ANDNOT LB403  ; P14 LoadIn Case3
ANDNOT LB404  ; P14 LoadIn Case4(DisCH)
ANDNOT LB405  ; P14 LoadIn Case5(DisCH)
ANDNOT LB406  ; P14 UnLoad Case1
ANDNOT LB407  ; P14 UnLoad Case2
ANDNOT LB408  ; P14 UnLoad Case3
ANDNOT LB409  ; P14 UnLoad Case4(DisCH)
ANDNOT LB410  ; P14 UnLoad Case5(DisCH)
LDNOT W199.00  ; DISCHARGE PROCESS START  // To protect conflict loop from dummy
ORNOT SHUTTER_DOOR_IN  ; CR.SHUTTER DOOR IN CONFIRM
ORNOT H41.00  ; DIAPH LOADER : LOADER STATUS1
ANDLD
OUT LB402  ; P14 LoadIn Case2
LD TR0
LD W93.02  ; Unit4CycleStartConditionAux3
OR LB403  ; P14 LoadIn Case3
ANDLD
ANDNOT LB401  ; P14 LoadIn Case1
ANDNOT LB402  ; P14 LoadIn Case2
ANDNOT LB404  ; P14 LoadIn Case4(DisCH)
ANDNOT LB405  ; P14 LoadIn Case5(DisCH)
ANDNOT LB406  ; P14 UnLoad Case1
ANDNOT LB407  ; P14 UnLoad Case2
ANDNOT LB408  ; P14 UnLoad Case3
ANDNOT LB409  ; P14 UnLoad Case4(DisCH)
ANDNOT LB410  ; P14 UnLoad Case5(DisCH)
OUT LB403  ; P14 LoadIn Case3
LD TR0
LD W93.03  ; Unit4CycleStartConditionAux4
OR LB404  ; P14 LoadIn Case4(DisCH)
ANDLD
ANDNOT LB401  ; P14 LoadIn Case1
ANDNOT LB402  ; P14 LoadIn Case2
ANDNOT LB403  ; P14 LoadIn Case3
ANDNOT LB405  ; P14 LoadIn Case5(DisCH)
ANDNOT LB406  ; P14 UnLoad Case1
ANDNOT LB407  ; P14 UnLoad Case2
ANDNOT LB408  ; P14 UnLoad Case3
ANDNOT LB409  ; P14 UnLoad Case4(DisCH)
ANDNOT LB410  ; P14 UnLoad Case5(DisCH)
OUT LB404  ; P14 LoadIn Case4(DisCH)
LD TR0
LD W93.04  ; Unit4CycleStartConditionAux5
OR LB405  ; P14 LoadIn Case5(DisCH)
ANDLD
ANDNOT LB401  ; P14 LoadIn Case1
ANDNOT LB402  ; P14 LoadIn Case2
ANDNOT LB403  ; P14 LoadIn Case3
ANDNOT LB404  ; P14 LoadIn Case4(DisCH)
ANDNOT LB406  ; P14 UnLoad Case1
ANDNOT LB407  ; P14 UnLoad Case2
ANDNOT LB408  ; P14 UnLoad Case3
ANDNOT LB409  ; P14 UnLoad Case4(DisCH)
ANDNOT LB410  ; P14 UnLoad Case5(DisCH)
OUT LB405  ; P14 LoadIn Case5(DisCH)

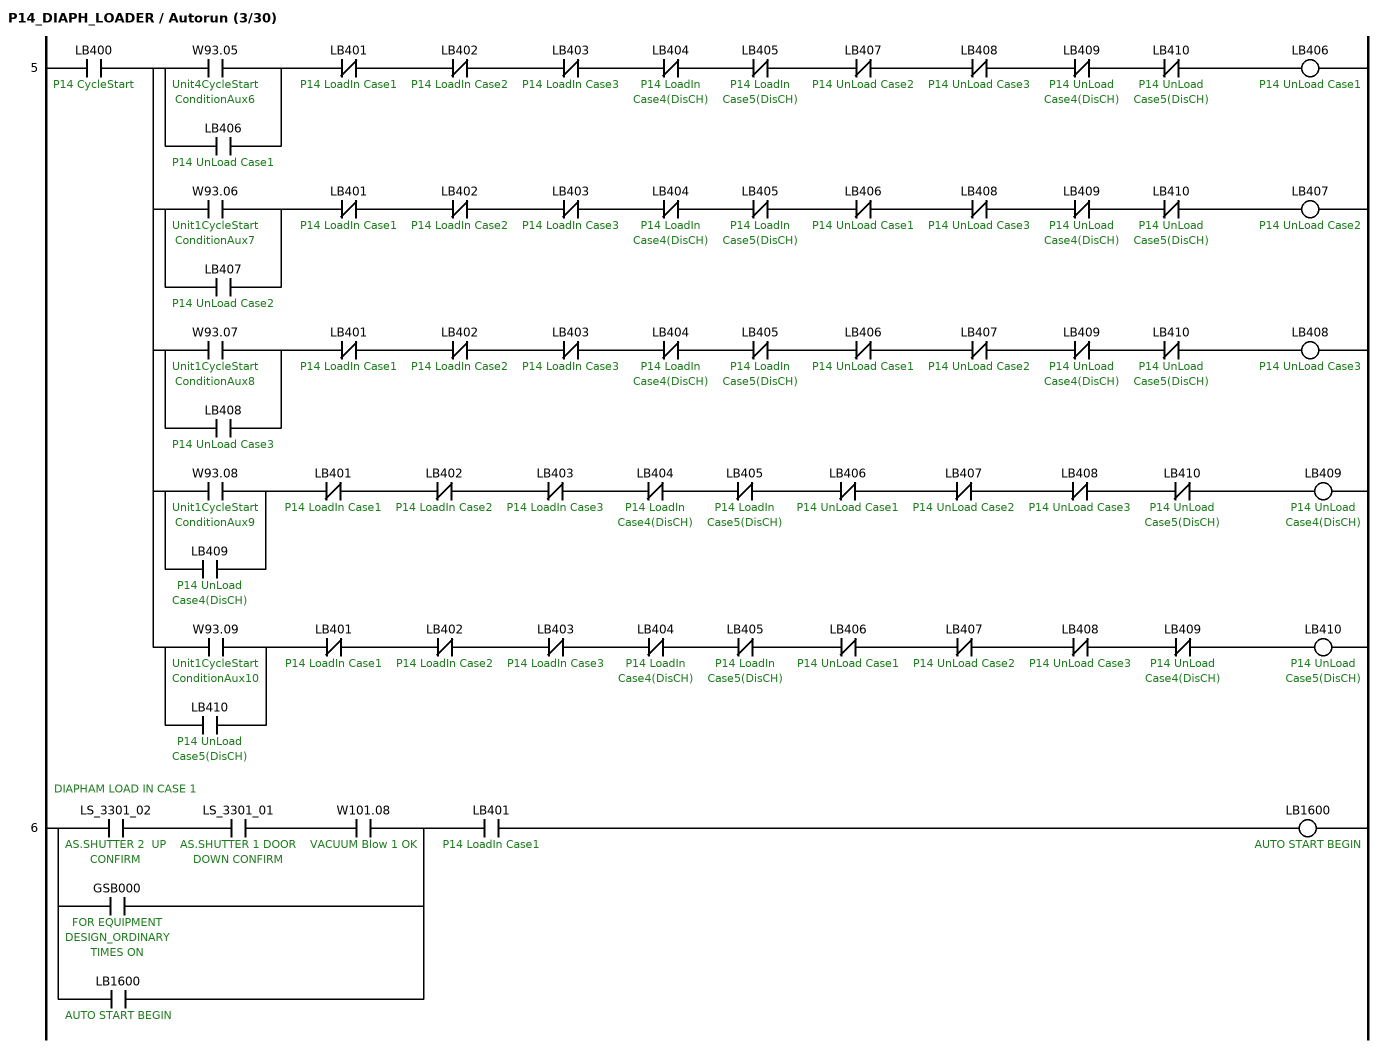
; rung 5
LD LB400  ; P14 CycleStart
OUT TR0
LD W93.05  ; Unit4CycleStartConditionAux6
OR LB406  ; P14 UnLoad Case1
ANDLD
ANDNOT LB401  ; P14 LoadIn Case1
ANDNOT LB402  ; P14 LoadIn Case2
ANDNOT LB403  ; P14 LoadIn Case3
ANDNOT LB404  ; P14 LoadIn Case4(DisCH)
ANDNOT LB405  ; P14 LoadIn Case5(DisCH)
ANDNOT LB407  ; P14 UnLoad Case2
ANDNOT LB408  ; P14 UnLoad Case3
ANDNOT LB409  ; P14 UnLoad Case4(DisCH)
ANDNOT LB410  ; P14 UnLoad Case5(DisCH)
OUT LB406  ; P14 UnLoad Case1
LD TR0
LD W93.06  ; Unit1CycleStartConditionAux7
OR LB407  ; P14 UnLoad Case2
ANDLD
ANDNOT LB401  ; P14 LoadIn Case1
ANDNOT LB402  ; P14 LoadIn Case2
ANDNOT LB403  ; P14 LoadIn Case3
ANDNOT LB404  ; P14 LoadIn Case4(DisCH)
ANDNOT LB405  ; P14 LoadIn Case5(DisCH)
ANDNOT LB406  ; P14 UnLoad Case1
ANDNOT LB408  ; P14 UnLoad Case3
ANDNOT LB409  ; P14 UnLoad Case4(DisCH)
ANDNOT LB410  ; P14 UnLoad Case5(DisCH)
OUT LB407  ; P14 UnLoad Case2
LD TR0
LD W93.07  ; Unit1CycleStartConditionAux8
OR LB408  ; P14 UnLoad Case3
ANDLD
ANDNOT LB401  ; P14 LoadIn Case1
ANDNOT LB402  ; P14 LoadIn Case2
ANDNOT LB403  ; P14 LoadIn Case3
ANDNOT LB404  ; P14 LoadIn Case4(DisCH)
ANDNOT LB405  ; P14 LoadIn Case5(DisCH)
ANDNOT LB406  ; P14 UnLoad Case1
ANDNOT LB407  ; P14 UnLoad Case2
ANDNOT LB409  ; P14 UnLoad Case4(DisCH)
ANDNOT LB410  ; P14 UnLoad Case5(DisCH)
OUT LB408  ; P14 UnLoad Case3
LD TR0
LD W93.08  ; Unit1CycleStartConditionAux9
OR LB409  ; P14 UnLoad Case4(DisCH)
ANDLD
ANDNOT LB401  ; P14 LoadIn Case1
ANDNOT LB402  ; P14 LoadIn Case2
ANDNOT LB403  ; P14 LoadIn Case3
ANDNOT LB404  ; P14 LoadIn Case4(DisCH)
ANDNOT LB405  ; P14 LoadIn Case5(DisCH)
ANDNOT LB406  ; P14 UnLoad Case1
ANDNOT LB407  ; P14 UnLoad Case2
ANDNOT LB408  ; P14 UnLoad Case3
ANDNOT LB410  ; P14 UnLoad Case5(DisCH)
OUT LB409  ; P14 UnLoad Case4(DisCH)
LD TR0
LD W93.09  ; Unit1CycleStartConditionAux10
OR LB410  ; P14 UnLoad Case5(DisCH)
ANDLD
ANDNOT LB401  ; P14 LoadIn Case1
ANDNOT LB402  ; P14 LoadIn Case2
ANDNOT LB403  ; P14 LoadIn Case3
ANDNOT LB404  ; P14 LoadIn Case4(DisCH)
ANDNOT LB405  ; P14 LoadIn Case5(DisCH)
ANDNOT LB406  ; P14 UnLoad Case1
ANDNOT LB407  ; P14 UnLoad Case2
ANDNOT LB408  ; P14 UnLoad Case3
ANDNOT LB409  ; P14 UnLoad Case4(DisCH)
OUT LB410  ; P14 UnLoad Case5(DisCH)
; rung 6: DIAPHAM LOAD IN CASE 1
LD LS_3301_02  ; AS.SHUTTER 2  UP CONFIRM
AND LS_3301_01  ; AS.SHUTTER 1 DOOR DOWN CONFIRM
AND W101.08  ; VACUUM Blow 1 OK
OR GSB000  ; FOR EQUIPMENT DESIGN_ORDINARY TIMES ON
OR LB1600  ; AUTO START BEGIN
AND LB401  ; P14 LoadIn Case1
OUT LB1600  ; AUTO START BEGIN

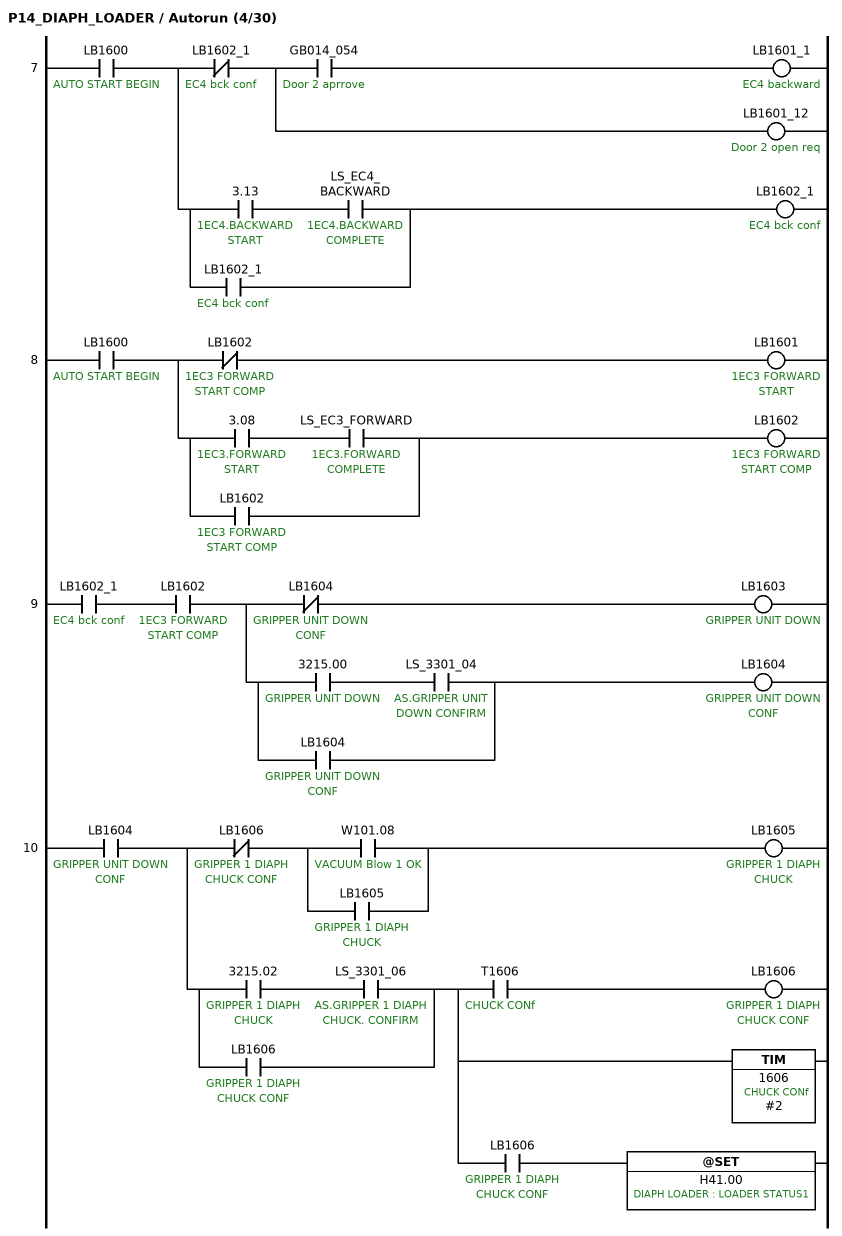
; rung 7
LD LB1600  ; AUTO START BEGIN
OUT TR0
ANDNOT LB1602_1  ; EC4 bck conf
OUT TR1
AND GB014_054  ; Door 2 aprrove
OUT LB1601_1  ; EC4 backward
LD TR1
OUT LB1601_12  ; Door 2 open req
LD TR0
LD 3.13  ; 1EC4.BACKWARD START
AND LS_EC4_BACKWARD  ; 1EC4.BACKWARD COMPLETE
OR LB1602_1  ; EC4 bck conf
ANDLD
OUT LB1602_1  ; EC4 bck conf
; rung 8
LD LB1600  ; AUTO START BEGIN
OUT TR0
ANDNOT LB1602  ; 1EC3 FORWARD START COMP
OUT LB1601  ; 1EC3 FORWARD START
LD TR0
LD 3.08  ; 1EC3.FORWARD START
AND LS_EC3_FORWARD  ; 1EC3.FORWARD COMPLETE
OR LB1602  ; 1EC3 FORWARD START COMP
ANDLD
OUT LB1602  ; 1EC3 FORWARD START COMP
; rung 9
LD LB1602_1  ; EC4 bck conf
AND LB1602  ; 1EC3 FORWARD START COMP
OUT TR0
ANDNOT LB1604  ; GRIPPER UNIT DOWN CONF
OUT LB1603  ; GRIPPER UNIT DOWN
LD TR0
LD 3215.00  ; GRIPPER UNIT DOWN
AND LS_3301_04  ; AS.GRIPPER UNIT DOWN CONFIRM
OR LB1604  ; GRIPPER UNIT DOWN CONF
ANDLD
OUT LB1604  ; GRIPPER UNIT DOWN CONF
; rung 10
LD LB1604  ; GRIPPER UNIT DOWN CONF
OUT TR0
ANDNOT LB1606  ; GRIPPER 1 DIAPH CHUCK CONF
LD W101.08  ; VACUUM Blow 1 OK
OR LB1605  ; GRIPPER 1 DIAPH CHUCK
ANDLD
OUT LB1605  ; GRIPPER 1 DIAPH CHUCK
LD TR0
LD 3215.02  ; GRIPPER 1 DIAPH CHUCK
AND LS_3301_06  ; AS.GRIPPER 1 DIAPH CHUCK. CONFIRM
OR LB1606  ; GRIPPER 1 DIAPH CHUCK CONF
ANDLD
OUT TR0
AND T1606  ; CHUCK CONf
OUT LB1606  ; GRIPPER 1 DIAPH CHUCK CONF
LD TR0
TIM 1606 #2  ; CHUCK CONf
AND LB1606  ; GRIPPER 1 DIAPH CHUCK CONF
@SET H41.00  ; DIAPH LOADER : LOADER STATUS1

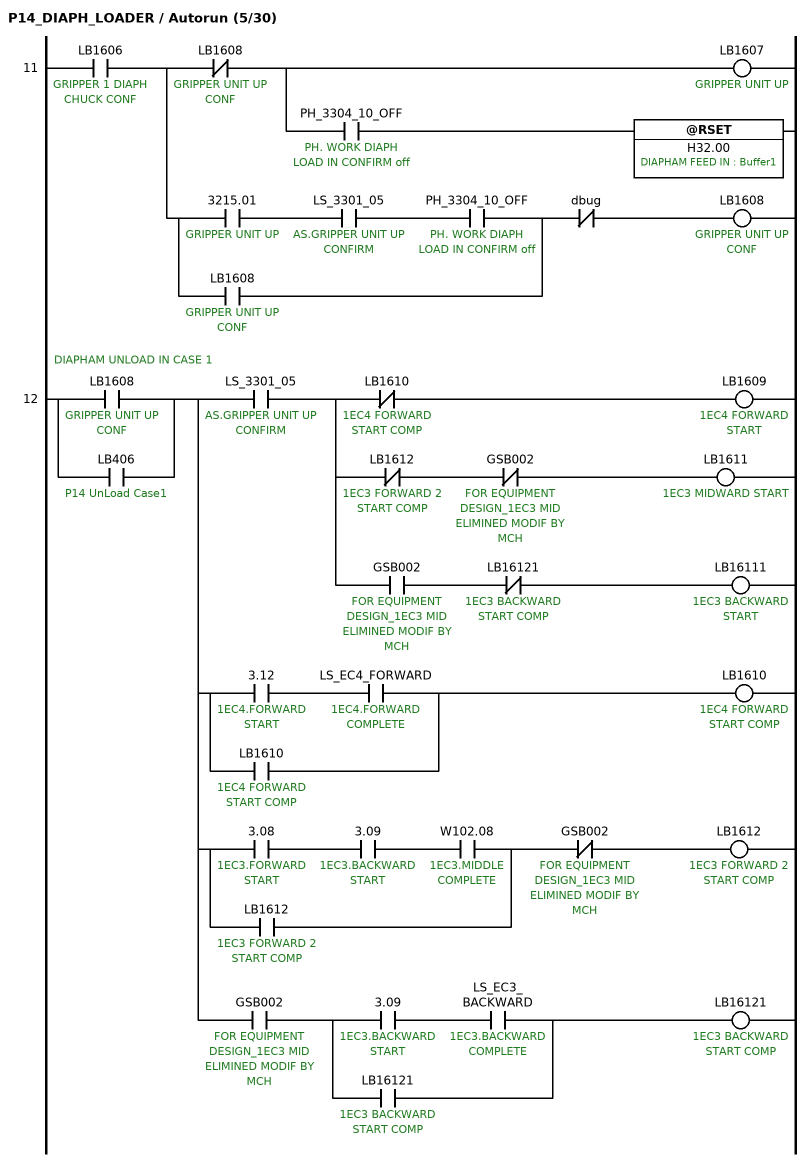
; rung 11
LD LB1606  ; GRIPPER 1 DIAPH CHUCK CONF
OUT TR0
ANDNOT LB1608  ; GRIPPER UNIT UP CONF
OUT LB1607  ; GRIPPER UNIT UP
AND PH_3304_10_OFF  ; PH. WORK DIAPH LOAD IN CONFIRM off
@RSET H32.00  ; DIAPHAM FEED IN : Buffer1
LD TR0
LD 3215.01  ; GRIPPER UNIT UP
AND LS_3301_05  ; AS.GRIPPER UNIT UP CONFIRM
AND PH_3304_10_OFF  ; PH. WORK DIAPH LOAD IN CONFIRM off
OR LB1608  ; GRIPPER UNIT UP CONF
ANDLD
ANDNOT dbug
OUT LB1608  ; GRIPPER UNIT UP CONF
; rung 12: DIAPHAM UNLOAD IN CASE 1
LD LB1608  ; GRIPPER UNIT UP CONF
OR LB406  ; P14 UnLoad Case1
OUT TR0
AND LS_3301_05  ; AS.GRIPPER UNIT UP CONFIRM
OUT TR1
ANDNOT LB1610  ; 1EC4 FORWARD START COMP
OUT LB1609  ; 1EC4 FORWARD START
LD TR1
ANDNOT LB1612  ; 1EC3 FORWARD 2 START COMP
ANDNOT GSB002  ; FOR EQUIPMENT DESIGN_1EC3 MID ELIMINED MODIF BY MCH
OUT LB1611  ; 1EC3 MIDWARD START
LD TR1
AND GSB002  ; FOR EQUIPMENT DESIGN_1EC3 MID ELIMINED MODIF BY MCH
ANDNOT LB16121  ; 1EC3 BACKWARD START COMP
OUT LB16111  ; 1EC3 BACKWARD START
LD TR0
LD 3.12  ; 1EC4.FORWARD START
AND LS_EC4_FORWARD  ; 1EC4.FORWARD COMPLETE
OR LB1610  ; 1EC4 FORWARD START COMP
ANDLD
OUT LB1610  ; 1EC4 FORWARD START COMP
LD TR0
LD 3.08  ; 1EC3.FORWARD START
AND 3.09  ; 1EC3.BACKWARD START
AND W102.08  ; 1EC3.MIDDLE COMPLETE
OR LB1612  ; 1EC3 FORWARD 2 START COMP
ANDLD
ANDNOT GSB002  ; FOR EQUIPMENT DESIGN_1EC3 MID ELIMINED MODIF BY MCH
OUT LB1612  ; 1EC3 FORWARD 2 START COMP
LD TR0
AND GSB002  ; FOR EQUIPMENT DESIGN_1EC3 MID ELIMINED MODIF BY MCH
LD 3.09  ; 1EC3.BACKWARD START
AND LS_EC3_BACKWARD  ; 1EC3.BACKWARD COMPLETE
OR LB16121  ; 1EC3 BACKWARD START COMP
ANDLD
OUT LB16121  ; 1EC3 BACKWARD START COMP

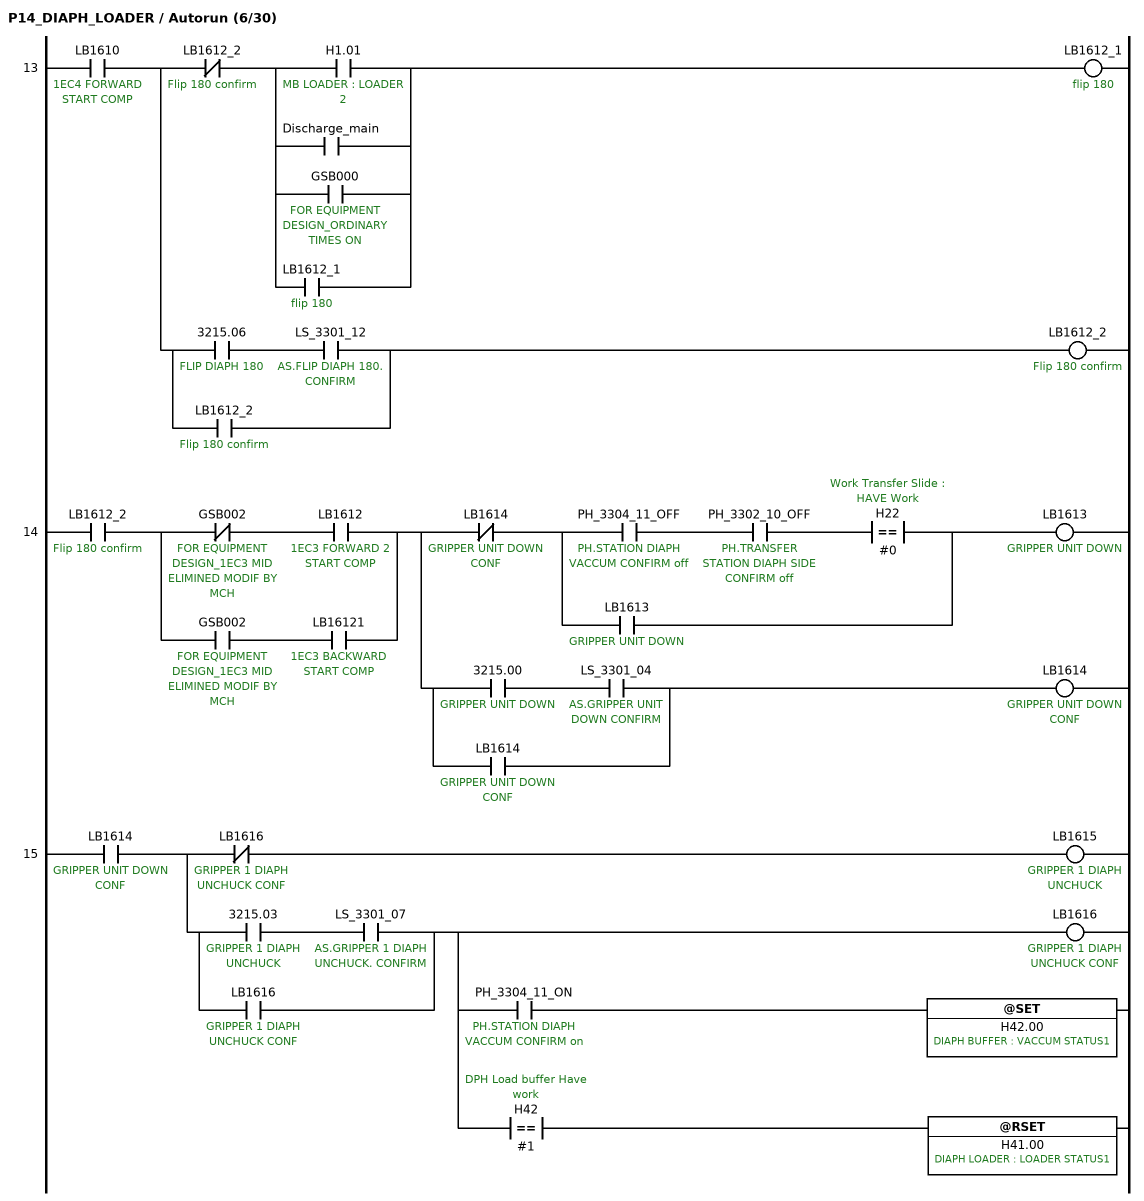
; rung 13
LD LB1610  ; 1EC4 FORWARD START COMP
OUT TR0
ANDNOT LB1612_2  ; Flip 180 confirm
LD H1.01  ; MB LOADER : LOADER 2
OR Discharge_main
OR GSB000  ; FOR EQUIPMENT DESIGN_ORDINARY TIMES ON
OR LB1612_1  ; flip 180
ANDLD
OUT LB1612_1  ; flip 180
LD TR0
LD 3215.06  ; FLIP DIAPH 180
AND LS_3301_12  ; AS.FLIP DIAPH 180. CONFIRM
OR LB1612_2  ; Flip 180 confirm
ANDLD
OUT LB1612_2  ; Flip 180 confirm
; rung 14
LD LB1612_2  ; Flip 180 confirm
LDNOT GSB002  ; FOR EQUIPMENT DESIGN_1EC3 MID ELIMINED MODIF BY MCH
AND LB1612  ; 1EC3 FORWARD 2 START COMP
LD GSB002  ; FOR EQUIPMENT DESIGN_1EC3 MID ELIMINED MODIF BY MCH
AND LB16121  ; 1EC3 BACKWARD START COMP
ORLD
ANDLD
OUT TR0
ANDNOT LB1614  ; GRIPPER UNIT DOWN CONF
LD PH_3304_11_OFF  ; PH.STATION DIAPH VACCUM CONFIRM off
AND PH_3302_10_OFF  ; PH.TRANSFER STATION DIAPH SIDE CONFIRM off
AND=(300) H22 #0  ; Work Transfer Slide : HAVE Work
OR LB1613  ; GRIPPER UNIT DOWN
ANDLD
OUT LB1613  ; GRIPPER UNIT DOWN
LD TR0
LD 3215.00  ; GRIPPER UNIT DOWN
AND LS_3301_04  ; AS.GRIPPER UNIT DOWN CONFIRM
OR LB1614  ; GRIPPER UNIT DOWN CONF
ANDLD
OUT LB1614  ; GRIPPER UNIT DOWN CONF
; rung 15
LD LB1614  ; GRIPPER UNIT DOWN CONF
OUT TR0
ANDNOT LB1616  ; GRIPPER 1 DIAPH UNCHUCK CONF
OUT LB1615  ; GRIPPER 1 DIAPH UNCHUCK
LD TR0
LD 3215.03  ; GRIPPER 1 DIAPH UNCHUCK
AND LS_3301_07  ; AS.GRIPPER 1 DIAPH UNCHUCK. CONFIRM
OR LB1616  ; GRIPPER 1 DIAPH UNCHUCK CONF
ANDLD
OUT TR0
OUT LB1616  ; GRIPPER 1 DIAPH UNCHUCK CONF
AND PH_3304_11_ON  ; PH.STATION DIAPH VACCUM CONFIRM on
@SET H42.00  ; DIAPH BUFFER : VACCUM STATUS1
LD TR0
AND=(300) H42 #1  ; DPH Load buffer Have work
@RSET H41.00  ; DIAPH LOADER : LOADER STATUS1

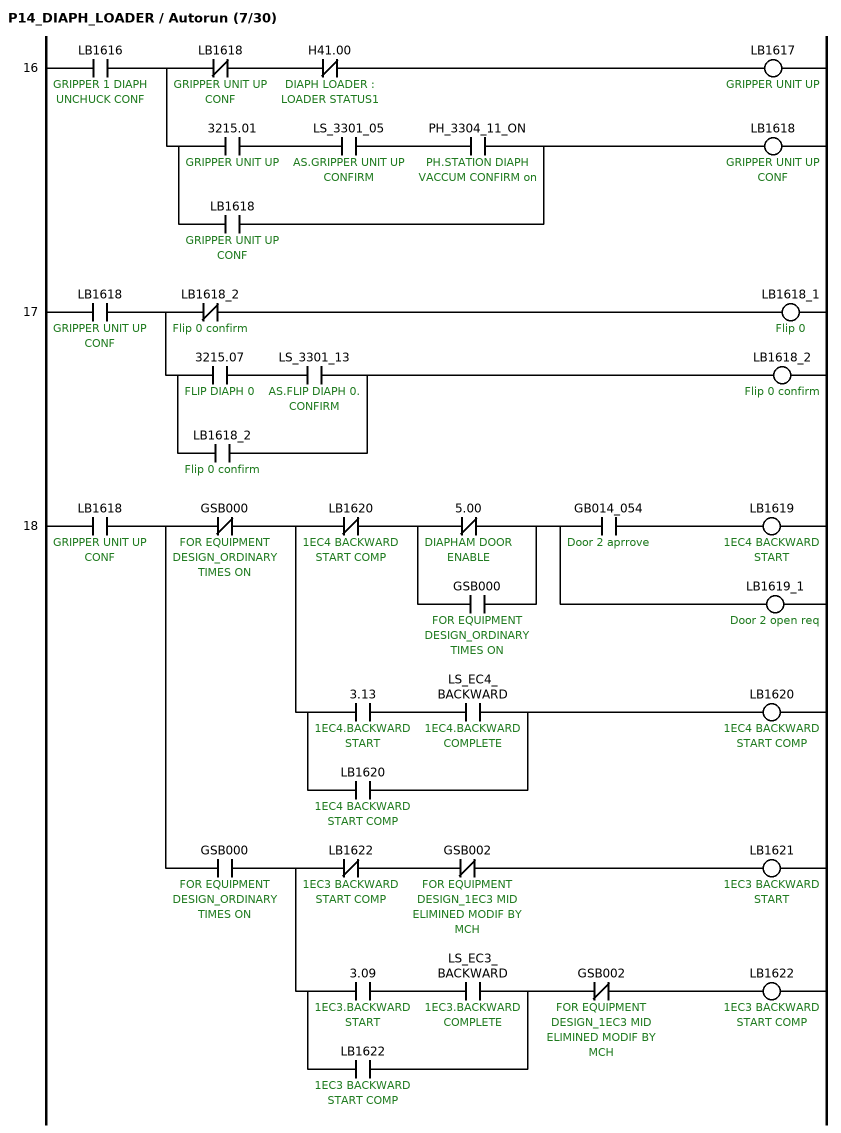
; rung 16
LD LB1616  ; GRIPPER 1 DIAPH UNCHUCK CONF
OUT TR0
ANDNOT LB1618  ; GRIPPER UNIT UP CONF
ANDNOT H41.00  ; DIAPH LOADER : LOADER STATUS1
OUT LB1617  ; GRIPPER UNIT UP
LD TR0
LD 3215.01  ; GRIPPER UNIT UP
AND LS_3301_05  ; AS.GRIPPER UNIT UP CONFIRM
AND PH_3304_11_ON  ; PH.STATION DIAPH VACCUM CONFIRM on
OR LB1618  ; GRIPPER UNIT UP CONF
ANDLD
OUT LB1618  ; GRIPPER UNIT UP CONF
; rung 17
LD LB1618  ; GRIPPER UNIT UP CONF
OUT TR0
ANDNOT LB1618_2  ; Flip 0 confirm
OUT LB1618_1  ; Flip 0
LD TR0
LD 3215.07  ; FLIP DIAPH 0
AND LS_3301_13  ; AS.FLIP DIAPH 0. CONFIRM
OR LB1618_2  ; Flip 0 confirm
ANDLD
OUT LB1618_2  ; Flip 0 confirm
; rung 18
LD LB1618  ; GRIPPER UNIT UP CONF
OUT TR0
ANDNOT GSB000  ; FOR EQUIPMENT DESIGN_ORDINARY TIMES ON
OUT TR1
ANDNOT LB1620  ; 1EC4 BACKWARD START COMP
LDNOT 5.00  ; DIAPHAM DOOR ENABLE
OR GSB000  ; FOR EQUIPMENT DESIGN_ORDINARY TIMES ON
ANDLD
OUT TR2
AND GB014_054  ; Door 2 aprrove
OUT LB1619  ; 1EC4 BACKWARD START
LD TR2
OUT LB1619_1  ; Door 2 open req
LD TR1
LD 3.13  ; 1EC4.BACKWARD START
AND LS_EC4_BACKWARD  ; 1EC4.BACKWARD COMPLETE
OR LB1620  ; 1EC4 BACKWARD START COMP
ANDLD
OUT LB1620  ; 1EC4 BACKWARD START COMP
LD TR0
AND GSB000  ; FOR EQUIPMENT DESIGN_ORDINARY TIMES ON
OUT TR0
ANDNOT LB1622  ; 1EC3 BACKWARD START COMP
ANDNOT GSB002  ; FOR EQUIPMENT DESIGN_1EC3 MID ELIMINED MODIF BY MCH
OUT LB1621  ; 1EC3 BACKWARD START
LD TR0
LD 3.09  ; 1EC3.BACKWARD START
AND LS_EC3_BACKWARD  ; 1EC3.BACKWARD COMPLETE
OR LB1622  ; 1EC3 BACKWARD START COMP
ANDLD
ANDNOT GSB002  ; FOR EQUIPMENT DESIGN_1EC3 MID ELIMINED MODIF BY MCH
OUT LB1622  ; 1EC3 BACKWARD START COMP

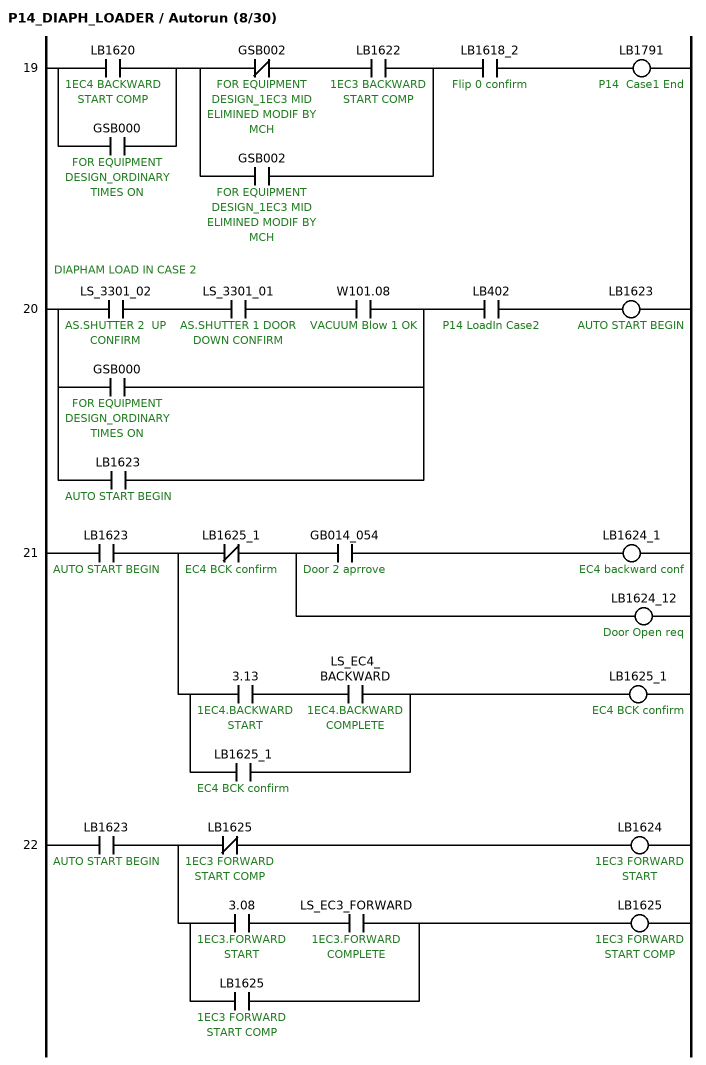
; rung 19
LD LB1620  ; 1EC4 BACKWARD START COMP
OR GSB000  ; FOR EQUIPMENT DESIGN_ORDINARY TIMES ON
LDNOT GSB002  ; FOR EQUIPMENT DESIGN_1EC3 MID ELIMINED MODIF BY MCH
AND LB1622  ; 1EC3 BACKWARD START COMP
OR GSB002  ; FOR EQUIPMENT DESIGN_1EC3 MID ELIMINED MODIF BY MCH
ANDLD
AND LB1618_2  ; Flip 0 confirm
OUT LB1791  ; P14  Case1 End
; rung 20: DIAPHAM LOAD IN CASE 2
LD LS_3301_02  ; AS.SHUTTER 2  UP CONFIRM
AND LS_3301_01  ; AS.SHUTTER 1 DOOR DOWN CONFIRM
AND W101.08  ; VACUUM Blow 1 OK
OR GSB000  ; FOR EQUIPMENT DESIGN_ORDINARY TIMES ON
OR LB1623  ; AUTO START BEGIN
AND LB402  ; P14 LoadIn Case2
OUT LB1623  ; AUTO START BEGIN
; rung 21
LD LB1623  ; AUTO START BEGIN
OUT TR0
ANDNOT LB1625_1  ; EC4 BCK confirm
OUT TR1
AND GB014_054  ; Door 2 aprrove
OUT LB1624_1  ; EC4 backward conf
LD TR1
OUT LB1624_12  ; Door Open req
LD TR0
LD 3.13  ; 1EC4.BACKWARD START
AND LS_EC4_BACKWARD  ; 1EC4.BACKWARD COMPLETE
OR LB1625_1  ; EC4 BCK confirm
ANDLD
OUT LB1625_1  ; EC4 BCK confirm
; rung 22
LD LB1623  ; AUTO START BEGIN
OUT TR0
ANDNOT LB1625  ; 1EC3 FORWARD START COMP
OUT LB1624  ; 1EC3 FORWARD START
LD TR0
LD 3.08  ; 1EC3.FORWARD START
AND LS_EC3_FORWARD  ; 1EC3.FORWARD COMPLETE
OR LB1625  ; 1EC3 FORWARD START COMP
ANDLD
OUT LB1625  ; 1EC3 FORWARD START COMP

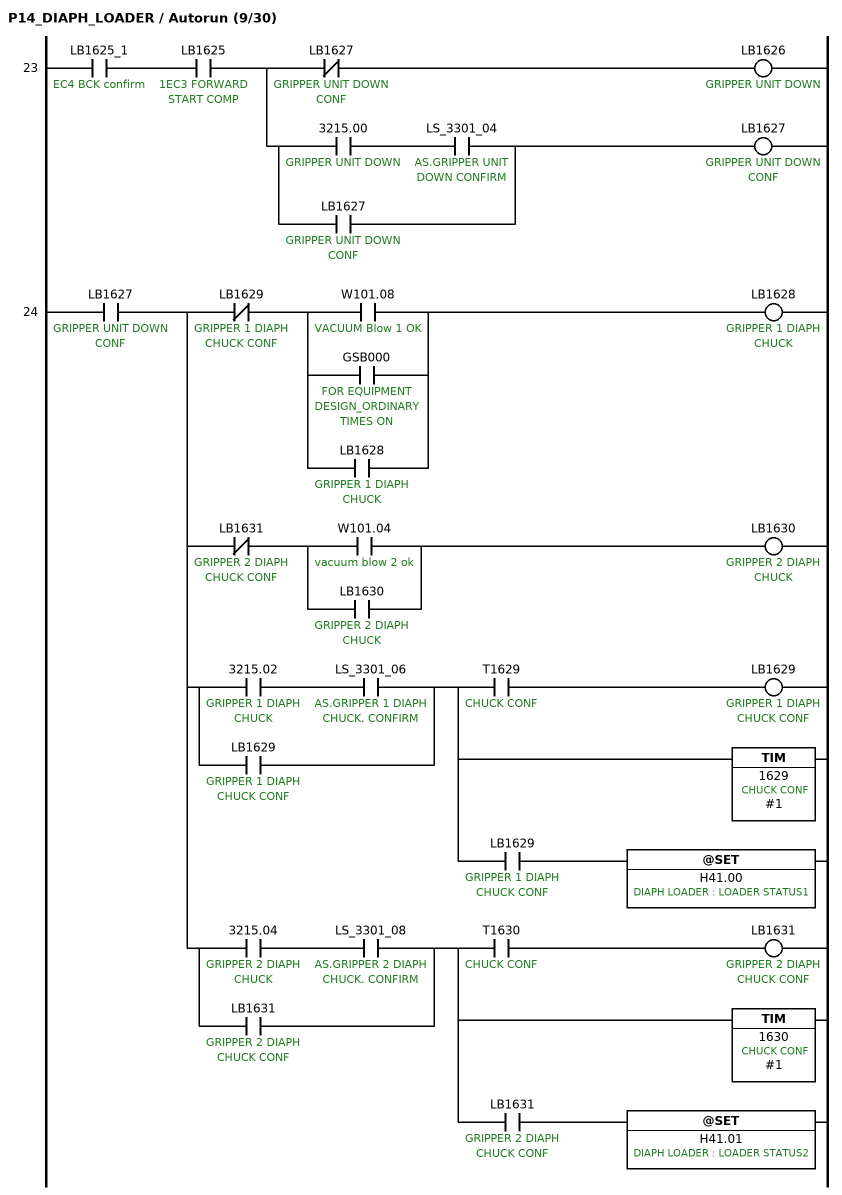
; rung 23
LD LB1625_1  ; EC4 BCK confirm
AND LB1625  ; 1EC3 FORWARD START COMP
OUT TR0
ANDNOT LB1627  ; GRIPPER UNIT DOWN CONF
OUT LB1626  ; GRIPPER UNIT DOWN
LD TR0
LD 3215.00  ; GRIPPER UNIT DOWN
AND LS_3301_04  ; AS.GRIPPER UNIT DOWN CONFIRM
OR LB1627  ; GRIPPER UNIT DOWN CONF
ANDLD
OUT LB1627  ; GRIPPER UNIT DOWN CONF
; rung 24
LD LB1627  ; GRIPPER UNIT DOWN CONF
OUT TR0
ANDNOT LB1629  ; GRIPPER 1 DIAPH CHUCK CONF
LD W101.08  ; VACUUM Blow 1 OK
OR GSB000  ; FOR EQUIPMENT DESIGN_ORDINARY TIMES ON
OR LB1628  ; GRIPPER 1 DIAPH CHUCK
ANDLD
OUT LB1628  ; GRIPPER 1 DIAPH CHUCK
LD TR0
ANDNOT LB1631  ; GRIPPER 2 DIAPH CHUCK CONF
LD W101.04  ; vacuum blow 2 ok
OR LB1630  ; GRIPPER 2 DIAPH CHUCK
ANDLD
OUT LB1630  ; GRIPPER 2 DIAPH CHUCK
LD TR0
LD 3215.02  ; GRIPPER 1 DIAPH CHUCK
AND LS_3301_06  ; AS.GRIPPER 1 DIAPH CHUCK. CONFIRM
OR LB1629  ; GRIPPER 1 DIAPH CHUCK CONF
ANDLD
OUT TR1
AND T1629  ; CHUCK CONF
OUT LB1629  ; GRIPPER 1 DIAPH CHUCK CONF
LD TR1
TIM 1629 #1  ; CHUCK CONF
AND LB1629  ; GRIPPER 1 DIAPH CHUCK CONF
@SET H41.00  ; DIAPH LOADER : LOADER STATUS1
LD TR0
LD 3215.04  ; GRIPPER 2 DIAPH CHUCK
AND LS_3301_08  ; AS.GRIPPER 2 DIAPH CHUCK. CONFIRM
OR LB1631  ; GRIPPER 2 DIAPH CHUCK CONF
ANDLD
OUT TR0
AND T1630  ; CHUCK CONF
OUT LB1631  ; GRIPPER 2 DIAPH CHUCK CONF
LD TR0
TIM 1630 #1  ; CHUCK CONF
AND LB1631  ; GRIPPER 2 DIAPH CHUCK CONF
@SET H41.01  ; DIAPH LOADER : LOADER STATUS2

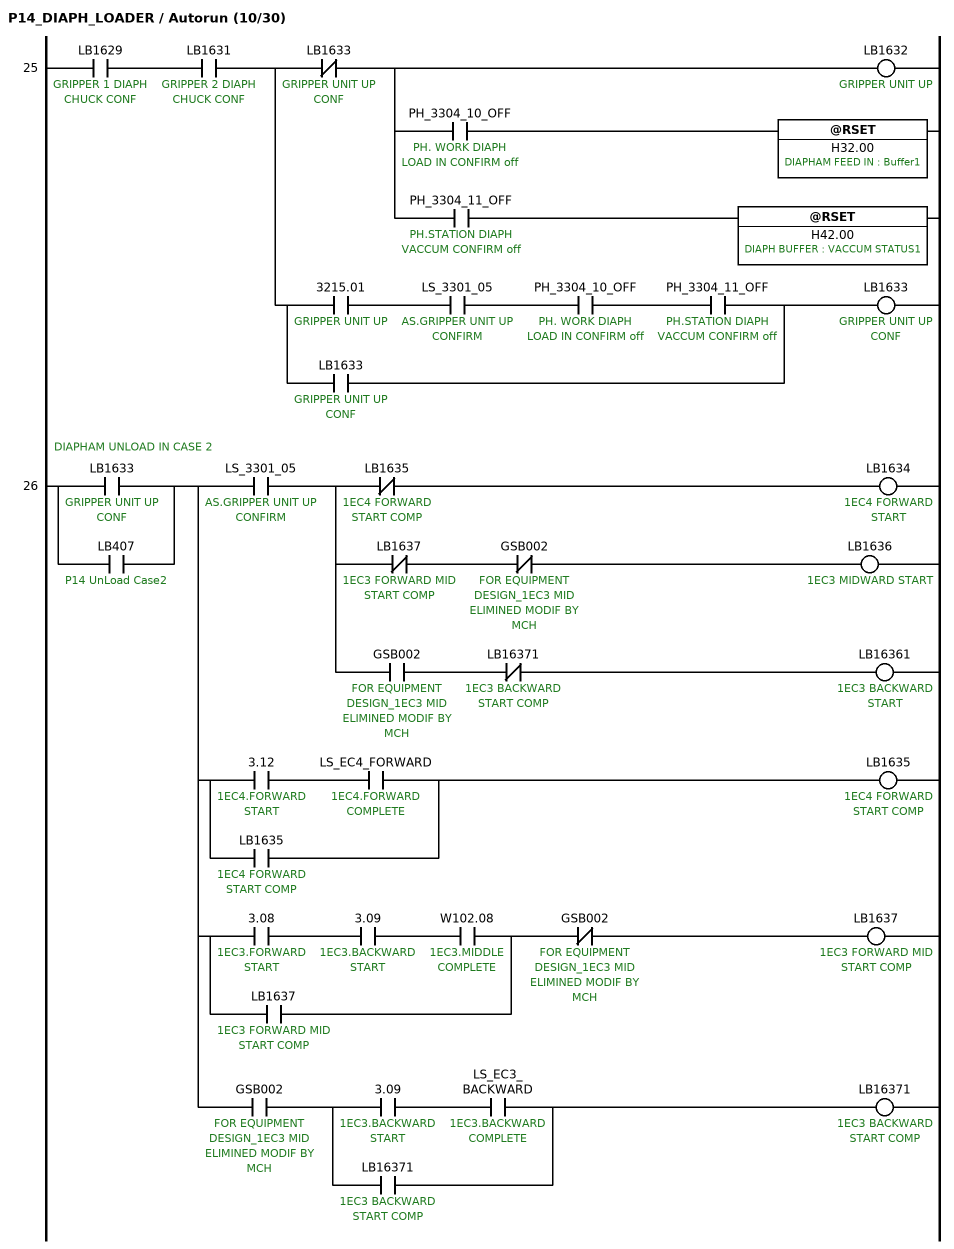
; rung 25
LD LB1629  ; GRIPPER 1 DIAPH CHUCK CONF
AND LB1631  ; GRIPPER 2 DIAPH CHUCK CONF
OUT TR0
ANDNOT LB1633  ; GRIPPER UNIT UP CONF
OUT TR1
OUT LB1632  ; GRIPPER UNIT UP
AND PH_3304_10_OFF  ; PH. WORK DIAPH LOAD IN CONFIRM off
@RSET H32.00  ; DIAPHAM FEED IN : Buffer1
LD TR1
AND PH_3304_11_OFF  ; PH.STATION DIAPH VACCUM CONFIRM off
@RSET H42.00  ; DIAPH BUFFER : VACCUM STATUS1
LD TR0
LD 3215.01  ; GRIPPER UNIT UP
AND LS_3301_05  ; AS.GRIPPER UNIT UP CONFIRM
AND PH_3304_10_OFF  ; PH. WORK DIAPH LOAD IN CONFIRM off
AND PH_3304_11_OFF  ; PH.STATION DIAPH VACCUM CONFIRM off
OR LB1633  ; GRIPPER UNIT UP CONF
ANDLD
OUT LB1633  ; GRIPPER UNIT UP CONF
; rung 26: DIAPHAM UNLOAD IN CASE 2
LD LB1633  ; GRIPPER UNIT UP CONF
OR LB407  ; P14 UnLoad Case2
OUT TR0
AND LS_3301_05  ; AS.GRIPPER UNIT UP CONFIRM
OUT TR1
ANDNOT LB1635  ; 1EC4 FORWARD START COMP
OUT LB1634  ; 1EC4 FORWARD START
LD TR1
ANDNOT LB1637  ; 1EC3 FORWARD MID START COMP
ANDNOT GSB002  ; FOR EQUIPMENT DESIGN_1EC3 MID ELIMINED MODIF BY MCH
OUT LB1636  ; 1EC3 MIDWARD START
LD TR1
AND GSB002  ; FOR EQUIPMENT DESIGN_1EC3 MID ELIMINED MODIF BY MCH
ANDNOT LB16371  ; 1EC3 BACKWARD START COMP
OUT LB16361  ; 1EC3 BACKWARD START
LD TR0
LD 3.12  ; 1EC4.FORWARD START
AND LS_EC4_FORWARD  ; 1EC4.FORWARD COMPLETE
OR LB1635  ; 1EC4 FORWARD START COMP
ANDLD
OUT LB1635  ; 1EC4 FORWARD START COMP
LD TR0
LD 3.08  ; 1EC3.FORWARD START
AND 3.09  ; 1EC3.BACKWARD START
AND W102.08  ; 1EC3.MIDDLE COMPLETE
OR LB1637  ; 1EC3 FORWARD MID START COMP
ANDLD
ANDNOT GSB002  ; FOR EQUIPMENT DESIGN_1EC3 MID ELIMINED MODIF BY MCH
OUT LB1637  ; 1EC3 FORWARD MID START COMP
LD TR0
AND GSB002  ; FOR EQUIPMENT DESIGN_1EC3 MID ELIMINED MODIF BY MCH
LD 3.09  ; 1EC3.BACKWARD START
AND LS_EC3_BACKWARD  ; 1EC3.BACKWARD COMPLETE
OR LB16371  ; 1EC3 BACKWARD START COMP
ANDLD
OUT LB16371  ; 1EC3 BACKWARD START COMP

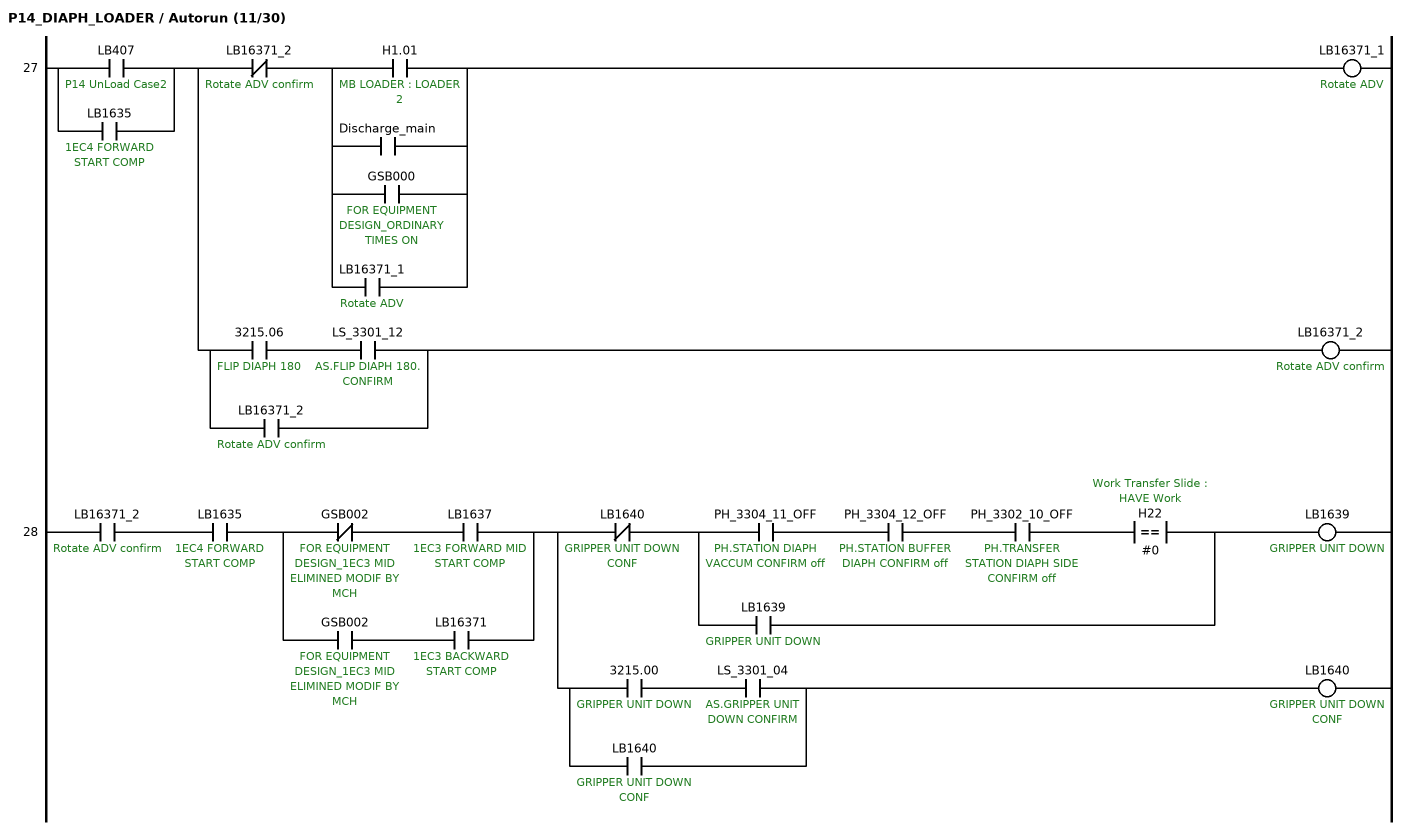
; rung 27
LD LB407  ; P14 UnLoad Case2
OR LB1635  ; 1EC4 FORWARD START COMP
OUT TR0
ANDNOT LB16371_2  ; Rotate ADV confirm
LD H1.01  ; MB LOADER : LOADER 2
OR Discharge_main
OR GSB000  ; FOR EQUIPMENT DESIGN_ORDINARY TIMES ON
OR LB16371_1  ; Rotate ADV
ANDLD
OUT LB16371_1  ; Rotate ADV
LD TR0
LD 3215.06  ; FLIP DIAPH 180
AND LS_3301_12  ; AS.FLIP DIAPH 180. CONFIRM
OR LB16371_2  ; Rotate ADV confirm
ANDLD
OUT LB16371_2  ; Rotate ADV confirm
; rung 28
LD LB16371_2  ; Rotate ADV confirm
AND LB1635  ; 1EC4 FORWARD START COMP
LDNOT GSB002  ; FOR EQUIPMENT DESIGN_1EC3 MID ELIMINED MODIF BY MCH
AND LB1637  ; 1EC3 FORWARD MID START COMP
LD GSB002  ; FOR EQUIPMENT DESIGN_1EC3 MID ELIMINED MODIF BY MCH
AND LB16371  ; 1EC3 BACKWARD START COMP
ORLD
ANDLD
OUT TR0
ANDNOT LB1640  ; GRIPPER UNIT DOWN CONF
LD PH_3304_11_OFF  ; PH.STATION DIAPH VACCUM CONFIRM off
AND PH_3304_12_OFF  ; PH.STATION BUFFER DIAPH CONFIRM off
AND PH_3302_10_OFF  ; PH.TRANSFER STATION DIAPH SIDE CONFIRM off
AND=(300) H22 #0  ; Work Transfer Slide : HAVE Work
OR LB1639  ; GRIPPER UNIT DOWN
ANDLD
OUT LB1639  ; GRIPPER UNIT DOWN
LD TR0
LD 3215.00  ; GRIPPER UNIT DOWN
AND LS_3301_04  ; AS.GRIPPER UNIT DOWN CONFIRM
OR LB1640  ; GRIPPER UNIT DOWN CONF
ANDLD
OUT LB1640  ; GRIPPER UNIT DOWN CONF

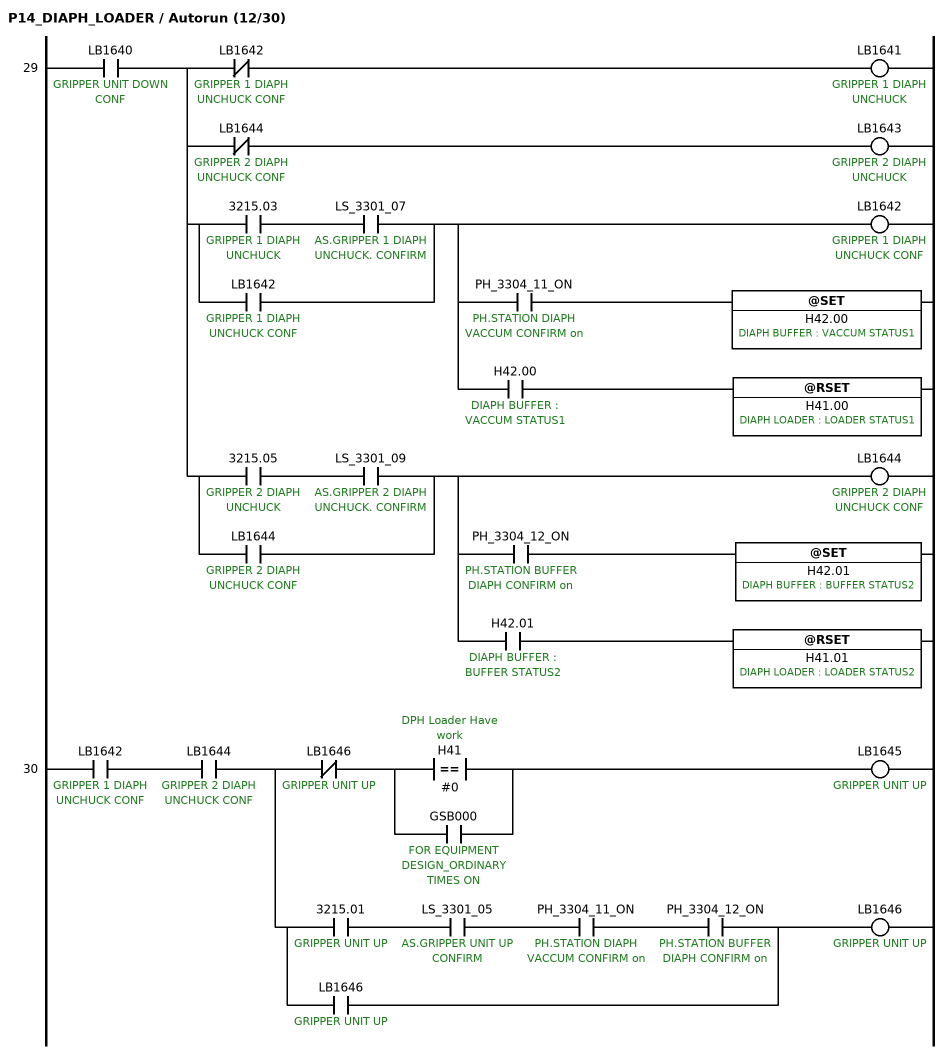
; rung 29
LD LB1640  ; GRIPPER UNIT DOWN CONF
OUT TR0
ANDNOT LB1642  ; GRIPPER 1 DIAPH UNCHUCK CONF
OUT LB1641  ; GRIPPER 1 DIAPH UNCHUCK
LD TR0
ANDNOT LB1644  ; GRIPPER 2 DIAPH UNCHUCK CONF
OUT LB1643  ; GRIPPER 2 DIAPH UNCHUCK
LD TR0
LD 3215.03  ; GRIPPER 1 DIAPH UNCHUCK
AND LS_3301_07  ; AS.GRIPPER 1 DIAPH UNCHUCK. CONFIRM
OR LB1642  ; GRIPPER 1 DIAPH UNCHUCK CONF
ANDLD
OUT TR1
OUT LB1642  ; GRIPPER 1 DIAPH UNCHUCK CONF
AND PH_3304_11_ON  ; PH.STATION DIAPH VACCUM CONFIRM on
@SET H42.00  ; DIAPH BUFFER : VACCUM STATUS1
LD TR1
AND H42.00  ; DIAPH BUFFER : VACCUM STATUS1
@RSET H41.00  ; DIAPH LOADER : LOADER STATUS1
LD TR0
LD 3215.05  ; GRIPPER 2 DIAPH UNCHUCK
AND LS_3301_09  ; AS.GRIPPER 2 DIAPH UNCHUCK. CONFIRM
OR LB1644  ; GRIPPER 2 DIAPH UNCHUCK CONF
ANDLD
OUT TR0
OUT LB1644  ; GRIPPER 2 DIAPH UNCHUCK CONF
AND PH_3304_12_ON  ; PH.STATION BUFFER DIAPH CONFIRM on
@SET H42.01  ; DIAPH BUFFER : BUFFER STATUS2
LD TR0
AND H42.01  ; DIAPH BUFFER : BUFFER STATUS2
@RSET H41.01  ; DIAPH LOADER : LOADER STATUS2
; rung 30
LD LB1642  ; GRIPPER 1 DIAPH UNCHUCK CONF
AND LB1644  ; GRIPPER 2 DIAPH UNCHUCK CONF
OUT TR0
ANDNOT LB1646  ; GRIPPER UNIT UP
LD=(300) H41 #0  ; DPH Loader Have work
OR GSB000  ; FOR EQUIPMENT DESIGN_ORDINARY TIMES ON
ANDLD
OUT LB1645  ; GRIPPER UNIT UP
LD TR0
LD 3215.01  ; GRIPPER UNIT UP
AND LS_3301_05  ; AS.GRIPPER UNIT UP CONFIRM
AND PH_3304_11_ON  ; PH.STATION DIAPH VACCUM CONFIRM on
AND PH_3304_12_ON  ; PH.STATION BUFFER DIAPH CONFIRM on
OR LB1646  ; GRIPPER UNIT UP
ANDLD
OUT LB1646  ; GRIPPER UNIT UP

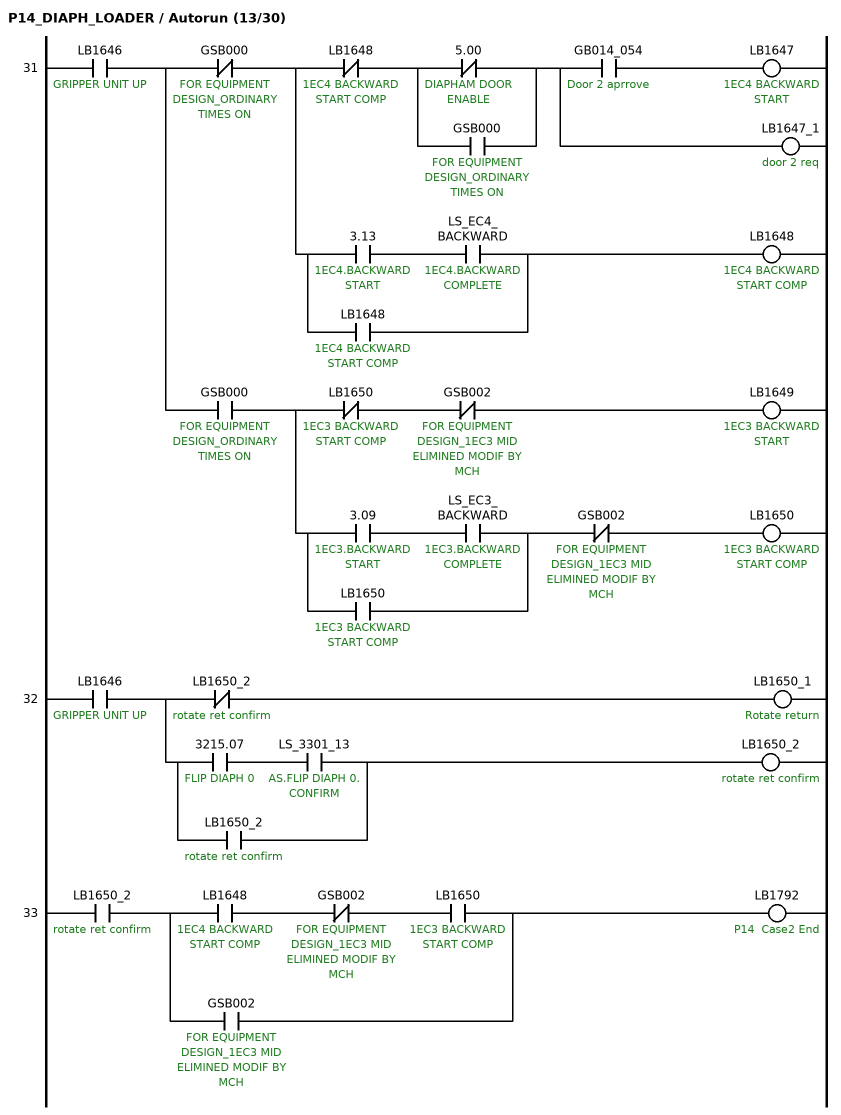
; rung 31
LD LB1646  ; GRIPPER UNIT UP
OUT TR0
ANDNOT GSB000  ; FOR EQUIPMENT DESIGN_ORDINARY TIMES ON
OUT TR1
ANDNOT LB1648  ; 1EC4 BACKWARD START COMP
LDNOT 5.00  ; DIAPHAM DOOR ENABLE
OR GSB000  ; FOR EQUIPMENT DESIGN_ORDINARY TIMES ON
ANDLD
OUT TR2
AND GB014_054  ; Door 2 aprrove
OUT LB1647  ; 1EC4 BACKWARD START
LD TR2
OUT LB1647_1  ; door 2 req
LD TR1
LD 3.13  ; 1EC4.BACKWARD START
AND LS_EC4_BACKWARD  ; 1EC4.BACKWARD COMPLETE
OR LB1648  ; 1EC4 BACKWARD START COMP
ANDLD
OUT LB1648  ; 1EC4 BACKWARD START COMP
LD TR0
AND GSB000  ; FOR EQUIPMENT DESIGN_ORDINARY TIMES ON
OUT TR0
ANDNOT LB1650  ; 1EC3 BACKWARD START COMP
ANDNOT GSB002  ; FOR EQUIPMENT DESIGN_1EC3 MID ELIMINED MODIF BY MCH
OUT LB1649  ; 1EC3 BACKWARD START
LD TR0
LD 3.09  ; 1EC3.BACKWARD START
AND LS_EC3_BACKWARD  ; 1EC3.BACKWARD COMPLETE
OR LB1650  ; 1EC3 BACKWARD START COMP
ANDLD
ANDNOT GSB002  ; FOR EQUIPMENT DESIGN_1EC3 MID ELIMINED MODIF BY MCH
OUT LB1650  ; 1EC3 BACKWARD START COMP
; rung 32
LD LB1646  ; GRIPPER UNIT UP
OUT TR0
ANDNOT LB1650_2  ; rotate ret confirm
OUT LB1650_1  ; Rotate return
LD TR0
LD 3215.07  ; FLIP DIAPH 0
AND LS_3301_13  ; AS.FLIP DIAPH 0. CONFIRM
OR LB1650_2  ; rotate ret confirm
ANDLD
OUT LB1650_2  ; rotate ret confirm
; rung 33
LD LB1650_2  ; rotate ret confirm
LD LB1648  ; 1EC4 BACKWARD START COMP
ANDNOT GSB002  ; FOR EQUIPMENT DESIGN_1EC3 MID ELIMINED MODIF BY MCH
AND LB1650  ; 1EC3 BACKWARD START COMP
OR GSB002  ; FOR EQUIPMENT DESIGN_1EC3 MID ELIMINED MODIF BY MCH
ANDLD
OUT LB1792  ; P14  Case2 End

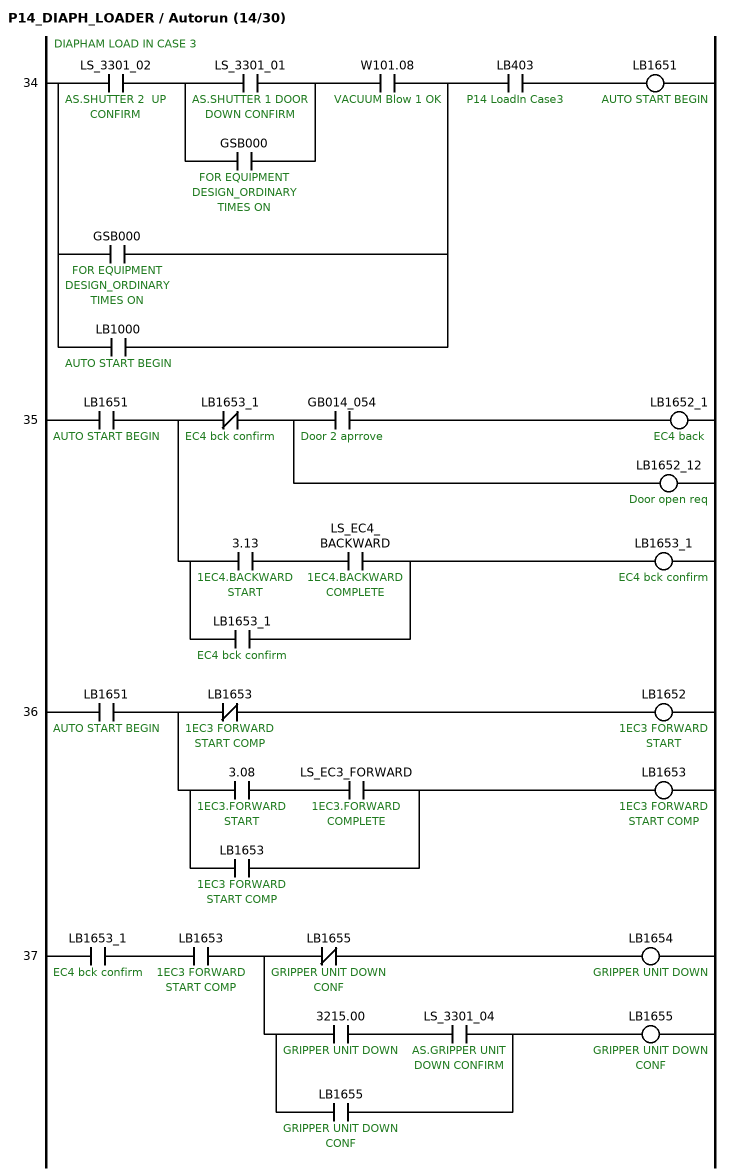
; rung 34: DIAPHAM LOAD IN CASE 3
LD LS_3301_02  ; AS.SHUTTER 2  UP CONFIRM
LD LS_3301_01  ; AS.SHUTTER 1 DOOR DOWN CONFIRM
OR GSB000  ; FOR EQUIPMENT DESIGN_ORDINARY TIMES ON
ANDLD
AND W101.08  ; VACUUM Blow 1 OK
OR GSB000  ; FOR EQUIPMENT DESIGN_ORDINARY TIMES ON
OR LB1000  ; AUTO START BEGIN
AND LB403  ; P14 LoadIn Case3
OUT LB1651  ; AUTO START BEGIN
; rung 35
LD LB1651  ; AUTO START BEGIN
OUT TR0
ANDNOT LB1653_1  ; EC4 bck confirm
OUT TR1
AND GB014_054  ; Door 2 aprrove
OUT LB1652_1  ; EC4 back
LD TR1
OUT LB1652_12  ; Door open req
LD TR0
LD 3.13  ; 1EC4.BACKWARD START
AND LS_EC4_BACKWARD  ; 1EC4.BACKWARD COMPLETE
OR LB1653_1  ; EC4 bck confirm
ANDLD
OUT LB1653_1  ; EC4 bck confirm
; rung 36
LD LB1651  ; AUTO START BEGIN
OUT TR0
ANDNOT LB1653  ; 1EC3 FORWARD START COMP
OUT LB1652  ; 1EC3 FORWARD START
LD TR0
LD 3.08  ; 1EC3.FORWARD START
AND LS_EC3_FORWARD  ; 1EC3.FORWARD COMPLETE
OR LB1653  ; 1EC3 FORWARD START COMP
ANDLD
OUT LB1653  ; 1EC3 FORWARD START COMP
; rung 37
LD LB1653_1  ; EC4 bck confirm
AND LB1653  ; 1EC3 FORWARD START COMP
OUT TR0
ANDNOT LB1655  ; GRIPPER UNIT DOWN CONF
OUT LB1654  ; GRIPPER UNIT DOWN
LD TR0
LD 3215.00  ; GRIPPER UNIT DOWN
AND LS_3301_04  ; AS.GRIPPER UNIT DOWN CONFIRM
OR LB1655  ; GRIPPER UNIT DOWN CONF
ANDLD
OUT LB1655  ; GRIPPER UNIT DOWN CONF

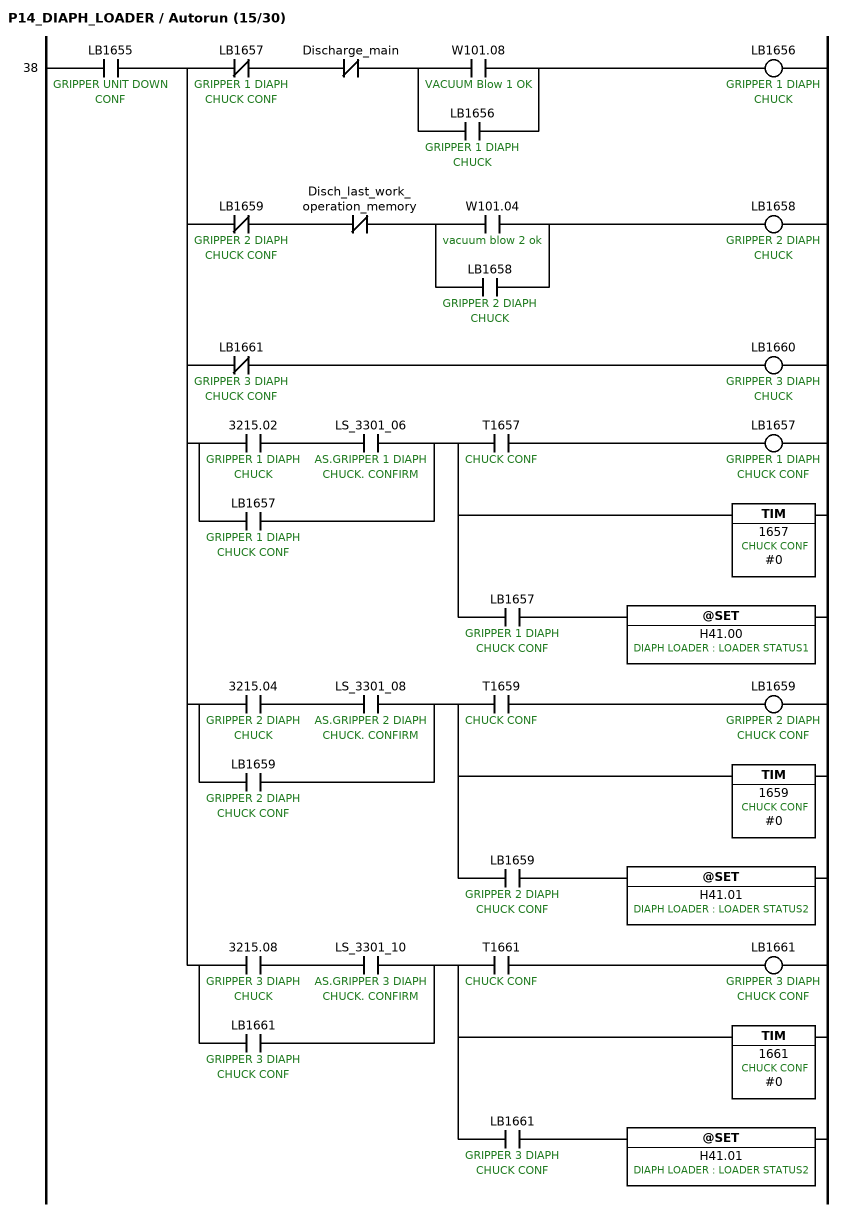
; rung 38
LD LB1655  ; GRIPPER UNIT DOWN CONF
OUT TR0
ANDNOT LB1657  ; GRIPPER 1 DIAPH CHUCK CONF
ANDNOT Discharge_main
LD W101.08  ; VACUUM Blow 1 OK
OR LB1656  ; GRIPPER 1 DIAPH CHUCK
ANDLD
OUT LB1656  ; GRIPPER 1 DIAPH CHUCK
LD TR0
ANDNOT LB1659  ; GRIPPER 2 DIAPH CHUCK CONF
ANDNOT Disch_last_work_operation_memory
LD W101.04  ; vacuum blow 2 ok
OR LB1658  ; GRIPPER 2 DIAPH CHUCK
ANDLD
OUT LB1658  ; GRIPPER 2 DIAPH CHUCK
LD TR0
ANDNOT LB1661  ; GRIPPER 3 DIAPH CHUCK CONF
OUT LB1660  ; GRIPPER 3 DIAPH CHUCK
LD TR0
LD 3215.02  ; GRIPPER 1 DIAPH CHUCK
AND LS_3301_06  ; AS.GRIPPER 1 DIAPH CHUCK. CONFIRM
OR LB1657  ; GRIPPER 1 DIAPH CHUCK CONF
ANDLD
OUT TR1
AND T1657  ; CHUCK CONF
OUT LB1657  ; GRIPPER 1 DIAPH CHUCK CONF
LD TR1
TIM 1657 #0  ; CHUCK CONF
AND LB1657  ; GRIPPER 1 DIAPH CHUCK CONF
@SET H41.00  ; DIAPH LOADER : LOADER STATUS1
LD TR0
LD 3215.04  ; GRIPPER 2 DIAPH CHUCK
AND LS_3301_08  ; AS.GRIPPER 2 DIAPH CHUCK. CONFIRM
OR LB1659  ; GRIPPER 2 DIAPH CHUCK CONF
ANDLD
OUT TR1
AND T1659  ; CHUCK CONF
OUT LB1659  ; GRIPPER 2 DIAPH CHUCK CONF
LD TR1
TIM 1659 #0  ; CHUCK CONF
AND LB1659  ; GRIPPER 2 DIAPH CHUCK CONF
@SET H41.01  ; DIAPH LOADER : LOADER STATUS2
LD TR0
LD 3215.08  ; GRIPPER 3 DIAPH CHUCK
AND LS_3301_10  ; AS.GRIPPER 3 DIAPH CHUCK. CONFIRM
OR LB1661  ; GRIPPER 3 DIAPH CHUCK CONF
ANDLD
OUT TR0
AND T1661  ; CHUCK CONF
OUT LB1661  ; GRIPPER 3 DIAPH CHUCK CONF
LD TR0
TIM 1661 #0  ; CHUCK CONF
AND LB1661  ; GRIPPER 3 DIAPH CHUCK CONF
@SET H41.01  ; DIAPH LOADER : LOADER STATUS2

